LIN {X 0,Y 235.015,Z 372.088,A -85,B 0,C 180,E1 -19772.385,E2 -19772.385} C_VEL
LIN {X 0,Y 234.992,Z 371.84,A -85,B 0,C 180,E1 -19775.247,E2 -19775.247} C_VEL
LIN {X 0,Y 235.016,Z 371.83,A -85,B 0,C 180,E1 -19778.97,E2 -19778.97} C_VEL
LIN {X 0,Y 235.101,Z 371.824,A -85,B 0,C 180,E1 -19783.059,E2 -19783.059} C_VEL
LIN {X 0,Y 235.152,Z 371.812,A -85,B 0,C 180,E1 -19787.924,E2 -19787.924} C_VEL
LIN {X 0,Y 235.395,Z 371.781,A -85,B 0,C 180,E1 -19791.414,E2 -19791.414} C_VEL
LIN {X 0,Y 235.411,Z 371.788,A -85,B 0,C 180,E1 -19793.141,E2 -19793.141} C_VEL
LIN {X 0,Y 235.6,Z 371.755,A -85,B 0,C 180,E1 -19798.29,E2 -19798.29} C_VEL
LIN {X 0,Y 235.6,Z 371.755,A -85,B 0,C 180,E1 -19801.709,E2 -19801.709} C_VEL
LIN {X 0,Y 235.372,Z 371.79,A -85,B 0,C 180,E1 -19806.859,E2 -19806.859} C_VEL
LIN {X 0,Y 235.218,Z 371.808,A -85,B 0,C 180,E1 -19810.327,E2 -19810.327} C_VEL
LIN {X 0,Y 235.118,Z 371.831,A -85,B 0,C 180,E1 -19815.606,E2 -19815.606} C_VEL
LIN {X 0,Y 235.022,Z 371.874,A -85,B 0,C 180,E1 -19819.658,E2 -19819.658} C_VEL
LIN {X 0,Y 235.358,Z 373.616,A -85,B 0,C 180,E1 -19822.842,E2 -19822.842} C_VEL
LIN {X 0,Y 235.843,Z 375.925,A -85,B 0,C 180,E1 -19826.62,E2 -19826.62} C_VEL
LIN {X 0,Y 236.341,Z 378.635,A -85,B 0,C 180,E1 -19830.416,E2 -19830.416} C_VEL
LIN {X 0,Y 236.912,Z 381.747,A -85,B 0,C 180,E1 -19834.307,E2 -19834.307} C_VEL
LIN {X 0,Y 237.605,Z 385.363,A -85,B 0,C 180,E1 -19838.4,E2 -19838.4} C_VEL
LIN {X 0,Y 238.386,Z 389.338,A -85,B 0,C 180,E1 -19842.519,E2 -19842.519} C_VEL
LIN {X 0,Y 238.664,Z 390.728,A -85,B 0,C 180,E1 -19843.886,E2 -19843.886} C_VEL
LIN {X 0,Y 238.895,Z 392.241,A -85,B 0,C 180,E1 -19844.731,E2 -19844.731} C_VEL
LIN {X 0,Y 239.346,Z 395.314,A -85,B 0,C 180,E1 -19845.625,E2 -19845.625} C_VEL
LIN {X 0,Y 240.189,Z 400.855,A -85,B 0,C 180,E1 -19846.595,E2 -19846.595} C_VEL
LIN {X 0,Y 243.299,Z 415.71,A -85,B 0,C 180,E1 -19848.361,E2 -19848.361} C_VEL
LIN {X 0,Y 244.82,Z 420.413,A -85,B 0,C 180,E1 -19849.055,E2 -19849.055} C_VEL
LIN {X 0,Y 247.249,Z 433.501,A -85,B 0,C 180,E1 -19850.799,E2 -19850.799} C_VEL
LIN {X 0,Y 248.739,Z 446.866,A -85,B 0,C 180,E1 -19852.698,E2 -19852.698} C_VEL
LIN {X 0,Y 249.245,Z 459.354,A -85,B 0,C 180,E1 -19854.629,E2 -19854.629} C_VEL
LIN {X 0,Y 248.915,Z 463.831,A -85,B 0,C 180,E1 -19855.336,E2 -19855.336} C_VEL
LIN {X 0,Y 245.212,Z 476.724,A -85,B 0,C 180,E1 -19857.249,E2 -19857.249} C_VEL
LIN {X 0,Y 241.61,Z 488.325,A -85,B 0,C 180,E1 -19859.399,E2 -19859.399} C_VEL
LIN {X 0,Y 238.108,Z 498.941,A -85,B 0,C 180,E1 -19861.819,E2 -19861.819} C_VEL
LIN {X 0,Y 235.174,Z 507.913,A -85,B 0,C 180,E1 -19864.321,E2 -19864.321} C_VEL
LIN {X 0,Y 232.556,Z 515.567,A -85,B 0,C 180,E1 -19866.866,E2 -19866.866} C_VEL
LIN {X 0,Y 230.383,Z 522.077,A -85,B 0,C 180,E1 -19869.462,E2 -19869.462} C_VEL
LIN {X 0,Y 228.333,Z 528.833,A -85,B 0,C 180,E1 -19872.78,E2 -19872.78} C_VEL
LIN {X 0,Y 226.762,Z 534.808,A -85,B 0,C 180,E1 -19876.559,E2 -19876.559} C_VEL
LIN {X 0,Y 226.093,Z 538.041,A -85,B 0,C 180,E1 -19879.251,E2 -19879.251} C_VEL
LIN {X 0,Y 225.715,Z 541.228,A -85,B 0,C 180,E1 -19882.845,E2 -19882.845} C_VEL
LIN {X 0,Y 225.73,Z 543.137,A -85,B 0,C 180,E1 -19886.43,E2 -19886.43} C_VEL
LIN {X 0,Y 225.822,Z 543.621,A -85,B 0,C 180,E1 -19888.216,E2 -19888.216} C_VEL
LIN {X 0,Y 225.878,Z 543.785,A -85,B 0,C 180,E1 -19890,E2 -19890} C_VEL
LIN {X 0,Y 225.823,Z 543.616,A -85,B 0,C 180,E1 -19891.783,E2 -19891.783} C_VEL
LIN {X 0,Y 225.741,Z 542.321,A -85,B 0,C 180,E1 -19895.359,E2 -19895.359} C_VEL
LIN {X 0,Y 225.869,Z 539.762,A -85,B 0,C 180,E1 -19898.95,E2 -19898.95} C_VEL
LIN {X 0,Y 226.451,Z 535.904,A -85,B 0,C 180,E1 -19902.547,E2 -19902.547} C_VEL
LIN {X 0,Y 227.762,Z 530.665,A -85,B 0,C 180,E1 -19906.124,E2 -19906.124} C_VEL
LIN {X 0,Y 229.759,Z 523.911,A -85,B 0,C 180,E1 -19909.662,E2 -19909.662} C_VEL
LIN {X 0,Y 232.12,Z 516.601,A -85,B 0,C 180,E1 -19912.708,E2 -19912.708} C_VEL
LIN {X 0,Y 235.14,Z 507.788,A -85,B 0,C 180,E1 -19915.683,E2 -19915.683} C_VEL
LIN {X 0,Y 238.097,Z 498.791,A -85,B 0,C 180,E1 -19918.182,E2 -19918.182} C_VEL
LIN {X 0,Y 241.563,Z 488.144,A -85,B 0,C 180,E1 -19920.607,E2 -19920.607} C_VEL
LIN {X 0,Y 245.156,Z 476.511,A -85,B 0,C 180,E1 -19922.759,E2 -19922.759} C_VEL
LIN {X 0,Y 248.879,Z 463.799,A -85,B 0,C 180,E1 -19924.63,E2 -19924.63} C_VEL
LIN {X 0,Y 249.127,Z 457.221,A -85,B 0,C 180,E1 -19925.672,E2 -19925.672} C_VEL
LIN {X 0,Y 248.45,Z 444.428,A -85,B 0,C 180,E1 -19927.623,E2 -19927.623} C_VEL
LIN {X 0,Y 246.857,Z 431.262,A -85,B 0,C 180,E1 -19929.47,E2 -19929.47} C_VEL
LIN {X 0,Y 244.147,Z 418.018,A -85,B 0,C 180,E1 -19931.234,E2 -19931.234} C_VEL
LIN {X 0,Y 241.259,Z 411.166,A -85,B 0,C 180,E1 -19932.337,E2 -19932.337} C_VEL
LIN {X 0,Y 236.412,Z 401.706,A -85,B 0,C 180,E1 -19933.98,E2 -19933.98} C_VEL
LIN {X 0,Y 234.193,Z 397.541,A -85,B 0,C 180,E1 -19934.687,E2 -19934.687} C_VEL
LIN {X 0,Y 232.289,Z 394.258,A -85,B 0,C 180,E1 -19935.292,E2 -19935.292} C_VEL
LIN {X 0,Y 231.858,Z 392.833,A -85,B 0,C 180,E1 -19935.518,E2 -19935.518} C_VEL
LIN {X 0,Y 231.002,Z 388.18,A -85,B 0,C 180,E1 -19940.29,E2 -19940.29} C_VEL
LIN {X 0,Y 230.054,Z 383.593,A -85,B 0,C 180,E1 -19945.572,E2 -19945.572} C_VEL
LIN {X 0,Y 229.331,Z 379.702,A -85,B 0,C 180,E1 -19950.638,E2 -19950.638} C_VEL
LIN {X 0,Y 228.852,Z 377.106,A -85,B 0,C 180,E1 -19954.537,E2 -19954.537} C_VEL
LIN {X 0,Y 228.397,Z 374.912,A -85,B 0,C 180,E1 -19958.331,E2 -19958.331} C_VEL
LIN {X 0,Y 228.04,Z 372.704,A -85,B 0,C 180,E1 -19962.823,E2 -19962.823} C_VEL
LIN {X 0,Y 228.076,Z 372.692,A -85,B 0,C 180,E1 -19967.544,E2 -19967.544} C_VEL
LIN {X 0,Y 228.266,Z 372.671,A -85,B 0,C 180,E1 -19971.145,E2 -19971.145} C_VEL
LIN {X 0,Y 228.322,Z 372.663,A -85,B 0,C 180,E1 -19972.928,E2 -19972.928} C_VEL
LIN {X 0,Y 228.557,Z 372.636,A -85,B 0,C 180,E1 -19978.238,E2 -19978.238} C_VEL
LIN {X 0,Y 228.557,Z 372.635,A -85,B 0,C 180,E1 -19981.762,E2 -19981.762} C_VEL
LIN {X 0,Y 228.362,Z 372.658,A -85,B 0,C 180,E1 -19987.072,E2 -19987.072} C_VEL
LIN {X 0,Y 228.175,Z 372.681,A -85,B 0,C 180,E1 -19990.65,E2 -19990.65} C_VEL
LIN {X 0,Y 228.069,Z 372.694,A -85,B 0,C 180,E1 -19994.272,E2 -19994.272} C_VEL
LIN {X 0,Y 228.006,Z 372.701,A -85,B 0,C 180,E1 -19997.953,E2 -19997.953} C_VEL
LIN {X 0,Y 227.933,Z 372.716,A -85,B 0,C 180,E1 -20002.33,E2 -20002.33} C_VEL
LIN {X 0,Y 227.946,Z 372.773,A -85,B 0,C 180,E1 -20005.084,E2 -20005.084} C_VEL
LIN {X 0,Y 228.303,Z 374.704,A -85,B 0,C 180,E1 -20009.508,E2 -20009.508} C_VEL
LIN {X 0,Y 228.687,Z 376.954,A -85,B 0,C 180,E1 -20013.925,E2 -20013.925} C_VEL
LIN {X 0,Y 229.075,Z 379.212,A -85,B 0,C 180,E1 -20017.851,E2 -20017.851} C_VEL
LIN {X 0,Y 229.499,Z 382.119,A -85,B 0,C 180,E1 -20022.355,E2 -20022.355} C_VEL
LIN {X 0,Y 229.854,Z 384.793,A -85,B 0,C 180,E1 -20026.131,E2 -20026.131} C_VEL
LIN {X 0,Y 229.888,Z 385.286,A -85,B 0,C 180,E1 -20026.793,E2 -20026.793} C_VEL
LIN {X 0,Y 231.265,Z 388.595,A -85,B 0,C 180,E1 -20027.302,E2 -20027.302} C_VEL
LIN {X 0,Y 232.899,Z 390.912,A -85,B 0,C 180,E1 -20027.804,E2 -20027.804} C_VEL
LIN {X 0,Y 237.12,Z 399.072,A -85,B 0,C 180,E1 -20029.257,E2 -20029.257} C_VEL
LIN {X 0,Y 241.328,Z 409.168,A -85,B 0,C 180,E1 -20030.956,E2 -20030.956} C_VEL
LIN {X 0,Y 245.03,Z 420.57,A -85,B 0,C 180,E1 -20032.812,E2 -20032.812} C_VEL
LIN {X 0,Y 247.842,Z 432.547,A -85,B 0,C 180,E1 -20034.79,E2 -20034.79} C_VEL
LIN {X 0,Y 249.545,Z 443.432,A -85,B 0,C 180,E1 -20036.689,E2 -20036.689} C_VEL
LIN {X 0,Y 250.061,Z 449.138,A -85,B 0,C 180,E1 -20037.724,E2 -20037.724} C_VEL
LIN {X 0,Y 247.163,Z 460.518,A -85,B 0,C 180,E1 -20039.451,E2 -20039.451} C_VEL
LIN {X 0,Y 244.196,Z 470.062,A -85,B 0,C 180,E1 -20041.179,E2 -20041.179} C_VEL
LIN {X 0,Y 240.769,Z 480.693,A -85,B 0,C 180,E1 -20043.567,E2 -20043.567} C_VEL
LIN {X 0,Y 237.529,Z 489.516,A -85,B 0,C 180,E1 -20045.994,E2 -20045.994} C_VEL
LIN {X 0,Y 234.851,Z 496.873,A -85,B 0,C 180,E1 -20048.487,E2 -20048.487} C_VEL
LIN {X 0,Y 232.143,Z 503.98,A -85,B 0,C 180,E1 -20051.465,E2 -20051.465} C_VEL
LIN {X 0,Y 229.682,Z 510.385,A -85,B 0,C 180,E1 -20054.925,E2 -20054.925} C_VEL
LIN {X 0,Y 227.926,Z 515.224,A -85,B 0,C 180,E1 -20058.438,E2 -20058.438} C_VEL
LIN {X 0,Y 227.059,Z 517.955,A -85,B 0,C 180,E1 -20061.097,E2 -20061.097} C_VEL
LIN {X 0,Y 226.328,Z 520.408,A -85,B 0,C 180,E1 -20064.655,E2 -20064.655} C_VEL
LIN {X 0,Y 225.966,Z 521.628,A -85,B 0,C 180,E1 -20068.218,E2 -20068.218} C_VEL
LIN {X 0,Y 225.965,Z 521.649,A -85,B 0,C 180,E1 -20071.783,E2 -20071.783} C_VEL
LIN {X 0,Y 226.317,Z 520.472,A -85,B 0,C 180,E1 -20075.346,E2 -20075.346} C_VEL
LIN {X 0,Y 226.992,Z 518.066,A -85,B 0,C 180,E1 -20078.906,E2 -20078.906} C_VEL
LIN {X 0,Y 228.275,Z 514.344,A -85,B 0,C 180,E1 -20082.446,E2 -20082.446} C_VEL
LIN {X 0,Y 230.161,Z 509.188,A -85,B 0,C 180,E1 -20085.951,E2 -20085.951} C_VEL
LIN {X 0,Y 232.106,Z 504.242,A -85,B 0,C 180,E1 -20088.538,E2 -20088.538} C_VEL
LIN {X 0,Y 234.807,Z 497.263,A -85,B 0,C 180,E1 -20091.488,E2 -20091.488} C_VEL
LIN {X 0,Y 237.423,Z 489.902,A -85,B 0,C 180,E1 -20094.018,E2 -20094.018} C_VEL
LIN {X 0,Y 240.657,Z 481.158,A -85,B 0,C 180,E1 -20096.446,E2 -20096.446} C_VEL
LIN {X 0,Y 244.11,Z 470.614,A -85,B 0,C 180,E1 -20098.832,E2 -20098.832} C_VEL
LIN {X 0,Y 247.705,Z 458.972,A -85,B 0,C 180,E1 -20100.921,E2 -20100.921} C_VEL
LIN {X 0,Y 250.104,Z 449.936,A -85,B 0,C 180,E1 -20102.27,E2 -20102.27} C_VEL
LIN {X 0,Y 249.142,Z 440.073,A -85,B 0,C 180,E1 -20104.042,E2 -20104.042} C_VEL
LIN {X 0,Y 247.061,Z 428.423,A -85,B 0,C 180,E1 -20106.02,E2 -20106.02} C_VEL
LIN {X 0,Y 243.944,Z 416.811,A -85,B 0,C 180,E1 -20107.937,E2 -20107.937} C_VEL
LIN {X 0,Y 239.95,Z 405.345,A -85,B 0,C 180,E1 -20109.811,E2 -20109.811} C_VEL
LIN {X 0,Y 235.604,Z 396.058,A -85,B 0,C 180,E1 -20111.422,E2 -20111.422} C_VEL
LIN {X 0,Y 232.307,Z 389.929,A -85,B 0,C 180,E1 -20112.542,E2 -20112.542} C_VEL
LIN {X 0,Y 230.416,Z 386.973,A -85,B 0,C 180,E1 -20113.145,E2 -20113.145} C_VEL
LIN {X 0,Y 229.888,Z 385.248,A -85,B 0,C 180,E1 -20113.423,E2 -20113.423} C_VEL
LIN {X 0,Y 229.514,Z 382.232,A -85,B 0,C 180,E1 -20117.649,E2 -20117.649} C_VEL
LIN {X 0,Y 229.081,Z 379.34,A -85,B 0,C 180,E1 -20122.151,E2 -20122.151} C_VEL
LIN {X 0,Y 228.711,Z 376.86,A -85,B 0,C 180,E1 -20126.418,E2 -20126.418} C_VEL
LIN {X 0,Y 228.339,Z 374.816,A -85,B 0,C 180,E1 -20130.497,E2 -20130.497} C_VEL
LIN {X 0,Y 227.964,Z 372.715,A -85,B 0,C 180,E1 -20135.344,E2 -20135.344} C_VEL
LIN {X 0,Y 227.966,Z 372.711,A -85,B 0,C 180,E1 -20138.287,E2 -20138.287} C_VEL
LIN {X 0,Y 228.039,Z 372.701,A -85,B 0,C 180,E1 -20142.825,E2 -20142.825} C_VEL
LIN {X 0,Y 228.099,Z 372.692,A -85,B 0,C 180,E1 -20147.544,E2 -20147.544} C_VEL
LIN {X 0,Y 228.33,Z 372.661,A -85,B 0,C 180,E1 -20151.147,E2 -20151.147} C_VEL
LIN {X 0,Y 228.363,Z 372.665,A -85,B 0,C 180,E1 -20152.928,E2 -20152.928} C_VEL
LIN {X 0,Y 228.559,Z 372.632,A -85,B 0,C 180,E1 -20158.238,E2 -20158.238} C_VEL
LIN {X 0,Y 228.558,Z 372.632,A -85,B 0,C 180,E1 -20161.762,E2 -20161.762} C_VEL
LIN {X 0,Y 228.322,Z 372.666,A -85,B 0,C 180,E1 -20167.072,E2 -20167.072} C_VEL
LIN {X 0,Y 228.154,Z 372.687,A -85,B 0,C 180,E1 -20170.65,E2 -20170.65} C_VEL
LIN {X 0,Y 228.069,Z 372.699,A -85,B 0,C 180,E1 -20174.271,E2 -20174.271} C_VEL
LIN {X 0,Y 228.05,Z 372.792,A -85,B 0,C 180,E1 -20177.184,E2 -20177.184} C_VEL
LIN {X 0,Y 228.434,Z 374.987,A -85,B 0,C 180,E1 -20181.665,E2 -20181.665} C_VEL
LIN {X 0,Y 228.886,Z 377.188,A -85,B 0,C 180,E1 -20185.459,E2 -20185.459} C_VEL
LIN {X 0,Y 229.361,Z 379.796,A -85,B 0,C 180,E1 -20189.358,E2 -20189.358} C_VEL
LIN {X 0,Y 230.068,Z 383.667,A -85,B 0,C 180,E1 -20194.433,E2 -20194.433} C_VEL
LIN {X 0,Y 230.591,Z 386.357,A -85,B 0,C 180,E1 -20197.585,E2 -20197.585} C_VEL
LIN {X 0,Y 231.386,Z 390.359,A -85,B 0,C 180,E1 -20201.929,E2 -20201.929} C_VEL
LIN {X 0,Y 231.861,Z 392.923,A -85,B 0,C 180,E1 -20204.48,E2 -20204.48} C_VEL
LIN {X 0,Y 233.212,Z 396.174,A -85,B 0,C 180,E1 -20204.951,E2 -20204.951} C_VEL
LIN {X 0,Y 234.925,Z 398.782,A -85,B 0,C 180,E1 -20205.478,E2 -20205.478} C_VEL
LIN {X 0,Y 241.608,Z 411.82,A -85,B 0,C 180,E1 -20207.727,E2 -20207.727} C_VEL
LIN {X 0,Y 243.299,Z 415.71,A -85,B 0,C 180,E1 -20208.361,E2 -20208.361} C_VEL
LIN {X 0,Y 244.001,Z 419.161,A -85,B 0,C 180,E1 -20208.777,E2 -20208.777} C_VEL
LIN {X 0,Y 244.156,Z 424.646,A -85,B 0,C 180,E1 -20209.308,E2 -20209.308} C_VEL
LIN {X 0,Y 242.658,Z 437.693,A -85,B 0,C 180,E1 -20210.463,E2 -20210.463} C_VEL
LIN {X 0,Y 242.29,Z 443.055,A -85,B 0,C 180,E1 -20211.089,E2 -20211.089} C_VEL
LIN {X 0,Y 242.378,Z 444.76,A -85,B 0,C 180,E1 -20211.333,E2 -20211.333} C_VEL
LIN {X 0,Y 242.974,Z 457.515,A -85,B 0,C 180,E1 -20213.361,E2 -20213.361} C_VEL
LIN {X 0,Y 242.891,Z 463.353,A -85,B 0,C 180,E1 -20214.347,E2 -20214.347} C_VEL
LIN {X 0,Y 240.378,Z 472.767,A -85,B 0,C 180,E1 -20215.749,E2 -20215.749} C_VEL
LIN {X 0,Y 236.768,Z 483.974,A -85,B 0,C 180,E1 -20217.703,E2 -20217.703} C_VEL
LIN {X 0,Y 232.983,Z 495.257,A -85,B 0,C 180,E1 -20220.15,E2 -20220.15} C_VEL
LIN {X 0,Y 229.694,Z 504.738,A -85,B 0,C 180,E1 -20222.68,E2 -20222.68} C_VEL
LIN {X 0,Y 226.471,Z 514.036,A -85,B 0,C 180,E1 -20225.72,E2 -20225.72} C_VEL
LIN {X 0,Y 223.63,Z 521.714,A -85,B 0,C 180,E1 -20228.813,E2 -20228.813} C_VEL
LIN {X 0,Y 221.33,Z 528.944,A -85,B 0,C 180,E1 -20232.486,E2 -20232.486} C_VEL
LIN {X 0,Y 219.779,Z 534.456,A -85,B 0,C 180,E1 -20236.123,E2 -20236.123} C_VEL
LIN {X 0,Y 219.069,Z 537.692,A -85,B 0,C 180,E1 -20238.902,E2 -20238.902} C_VEL
LIN {X 0,Y 218.628,Z 540.881,A -85,B 0,C 180,E1 -20242.612,E2 -20242.612} C_VEL
LIN {X 0,Y 218.64,Z 542.791,A -85,B 0,C 180,E1 -20246.314,E2 -20246.314} C_VEL
LIN {X 0,Y 218.809,Z 543.44,A -85,B 0,C 180,E1 -20250,E2 -20250} C_VEL
LIN {X 0,Y 218.731,Z 543.271,A -85,B 0,C 180,E1 -20251.841,E2 -20251.841} C_VEL
LIN {X 0,Y 218.647,Z 541.974,A -85,B 0,C 180,E1 -20255.533,E2 -20255.533} C_VEL
LIN {X 0,Y 218.796,Z 539.413,A -85,B 0,C 180,E1 -20259.242,E2 -20259.242} C_VEL
LIN {X 0,Y 219.467,Z 535.553,A -85,B 0,C 180,E1 -20262.953,E2 -20262.953} C_VEL
LIN {X 0,Y 220.854,Z 530.309,A -85,B 0,C 180,E1 -20266.642,E2 -20266.642} C_VEL
LIN {X 0,Y 222.991,Z 523.55,A -85,B 0,C 180,E1 -20270.285,E2 -20270.285} C_VEL
LIN {X 0,Y 225.527,Z 516.235,A -85,B 0,C 180,E1 -20273.411,E2 -20273.411} C_VEL
LIN {X 0,Y 228.695,Z 507.412,A -85,B 0,C 180,E1 -20276.462,E2 -20276.462} C_VEL
LIN {X 0,Y 232.34,Z 496.75,A -85,B 0,C 180,E1 -20279.442,E2 -20279.442} C_VEL
LIN {X 0,Y 236.114,Z 485.771,A -85,B 0,C 180,E1 -20281.893,E2 -20281.893} C_VEL
LIN {X 0,Y 239.579,Z 474.902,A -85,B 0,C 180,E1 -20283.874,E2 -20283.874} C_VEL
LIN {X 0,Y 242.646,Z 464.741,A -85,B 0,C 180,E1 -20285.4,E2 -20285.4} C_VEL
LIN {X 0,Y 242.904,Z 455.67,A -85,B 0,C 180,E1 -20286.896,E2 -20286.896} C_VEL
LIN {X 0,Y 242.101,Z 442.227,A -85,B 0,C 180,E1 -20288.997,E2 -20288.997} C_VEL
LIN {X 0,Y 240.271,Z 428.605,A -85,B 0,C 180,E1 -20290.97,E2 -20290.97} C_VEL
LIN {X 0,Y 238.358,Z 420.17,A -85,B 0,C 180,E1 -20292.189,E2 -20292.189} C_VEL
LIN {X 0,Y 233.484,Z 409.417,A -85,B 0,C 180,E1 -20294.135,E2 -20294.135} C_VEL
LIN {X 0,Y 229.654,Z 402.034,A -85,B 0,C 180,E1 -20295.519,E2 -20295.519} C_VEL
LIN {X 0,Y 227.202,Z 397.587,A -85,B 0,C 180,E1 -20296.359,E2 -20296.359} C_VEL
LIN {X 0,Y 225.212,Z 394.558,A -85,B 0,C 180,E1 -20297.027,E2 -20297.027} C_VEL
LIN {X 0,Y 224.567,Z 392.591,A -85,B 0,C 180,E1 -20297.333,E2 -20297.333} C_VEL
LIN {X 0,Y 223.899,Z 389.135,A -85,B 0,C 180,E1 -20301.114,E2 -20301.114} C_VEL
LIN {X 0,Y 223.225,Z 385.48,A -85,B 0,C 180,E1 -20305.479,E2 -20305.479} C_VEL
LIN {X 0,Y 222.612,Z 382.328,A -85,B 0,C 180,E1 -20309.66,E2 -20309.66} C_VEL
LIN {X 0,Y 222.129,Z 379.615,A -85,B 0,C 180,E1 -20313.708,E2 -20313.708} C_VEL
LIN {X 0,Y 221.694,Z 377.313,A -85,B 0,C 180,E1 -20317.641,E2 -20317.641} C_VEL
LIN {X 0,Y 221.213,Z 374.557,A -85,B 0,C 180,E1 -20323.386,E2 -20323.386} C_VEL
LIN {X 0,Y 221.007,Z 373.575,A -85,B 0,C 180,E1 -20326.202,E2 -20326.202} C_VEL
LIN {X 0,Y 221.204,Z 373.549,A -85,B 0,C 180,E1 -20330.86,E2 -20330.86} C_VEL
LIN {X 0,Y 221.141,Z 373.558,A -85,B 0,C 180,E1 -20334.529,E2 -20334.529} C_VEL
LIN {X 0,Y 221.515,Z 373.513,A -85,B 0,C 180,E1 -20338.182,E2 -20338.182} C_VEL
LIN {X 0,Y 221.515,Z 373.513,A -85,B 0,C 180,E1 -20341.818,E2 -20341.818} C_VEL
LIN {X 0,Y 221.299,Z 373.536,A -85,B 0,C 180,E1 -20347.298,E2 -20347.298} C_VEL
LIN {X 0,Y 221.12,Z 373.558,A -85,B 0,C 180,E1 -20350.994,E2 -20350.994} C_VEL
LIN {X 0,Y 221.02,Z 373.58,A -85,B 0,C 180,E1 -20356.63,E2 -20356.63} C_VEL
LIN {X 0,Y 220.907,Z 373.635,A -85,B 0,C 180,E1 -20362.198,E2 -20362.198} C_VEL
LIN {X 0,Y 221.21,Z 375.203,A -85,B 0,C 180,E1 -20366.41,E2 -20366.41} C_VEL
LIN {X 0,Y 221.553,Z 377.285,A -85,B 0,C 180,E1 -20371.076,E2 -20371.076} C_VEL
LIN {X 0,Y 221.881,Z 379.157,A -85,B 0,C 180,E1 -20374.761,E2 -20374.761} C_VEL
LIN {X 0,Y 222.167,Z 380.841,A -85,B 0,C 180,E1 -20377.735,E2 -20377.735} C_VEL
LIN {X 0,Y 222.487,Z 383.225,A -85,B 0,C 180,E1 -20381.557,E2 -20381.557} C_VEL
LIN {X 0,Y 222.921,Z 385.725,A -85,B 0,C 180,E1 -20385.023,E2 -20385.023} C_VEL
LIN {X 0,Y 224.353,Z 388.977,A -85,B 0,C 180,E1 -20385.576,E2 -20385.576} C_VEL
LIN {X 0,Y 225.895,Z 390.967,A -85,B 0,C 180,E1 -20386.081,E2 -20386.081} C_VEL
LIN {X 0,Y 228.091,Z 394.897,A -85,B 0,C 180,E1 -20386.876,E2 -20386.876} C_VEL
LIN {X 0,Y 232.253,Z 403.056,A -85,B 0,C 180,E1 -20388.464,E2 -20388.464} C_VEL
LIN {X 0,Y 236.139,Z 412.811,A -85,B 0,C 180,E1 -20390.195,E2 -20390.195} C_VEL
LIN {X 0,Y 239.781,Z 425.003,A -85,B 0,C 180,E1 -20392.314,E2 -20392.314} C_VEL
LIN {X 0,Y 242.16,Z 436.585,A -85,B 0,C 180,E1 -20394.353,E2 -20394.353} C_VEL
LIN {X 0,Y 243.584,Z 447.83,A -85,B 0,C 180,E1 -20396.434,E2 -20396.434} C_VEL
LIN {X 0,Y 243.841,Z 450.945,A -85,B 0,C 180,E1 -20397.029,E2 -20397.029} C_VEL
LIN {X 0,Y 240.444,Z 463.235,A -85,B 0,C 180,E1 -20398.991,E2 -20398.991} C_VEL
LIN {X 0,Y 237.391,Z 472.402,A -85,B 0,C 180,E1 -20400.759,E2 -20400.759} C_VEL
LIN {X 0,Y 233.843,Z 482.688,A -85,B 0,C 180,E1 -20403.204,E2 -20403.204} C_VEL
LIN {X 0,Y 230.544,Z 491.22,A -85,B 0,C 180,E1 -20405.698,E2 -20405.698} C_VEL
LIN {X 0,Y 227.842,Z 498.346,A -85,B 0,C 180,E1 -20408.275,E2 -20408.275} C_VEL
LIN {X 0,Y 225.428,Z 504.335,A -85,B 0,C 180,E1 -20410.892,E2 -20410.892} C_VEL
LIN {X 0,Y 222.828,Z 510.737,A -85,B 0,C 180,E1 -20414.449,E2 -20414.449} C_VEL
LIN {X 0,Y 220.983,Z 515.572,A -85,B 0,C 180,E1 -20418.07,E2 -20418.07} C_VEL
LIN {X 0,Y 220.039,Z 518.302,A -85,B 0,C 180,E1 -20420.811,E2 -20420.811} C_VEL
LIN {X 0,Y 219.277,Z 520.753,A -85,B 0,C 180,E1 -20424.482,E2 -20424.482} C_VEL
LIN {X 0,Y 218.901,Z 521.973,A -85,B 0,C 180,E1 -20428.16,E2 -20428.16} C_VEL
LIN {X 0,Y 218.901,Z 521.992,A -85,B 0,C 180,E1 -20431.84,E2 -20431.84} C_VEL
LIN {X 0,Y 219.264,Z 520.817,A -85,B 0,C 180,E1 -20435.518,E2 -20435.518} C_VEL
LIN {X 0,Y 219.994,Z 518.411,A -85,B 0,C 180,E1 -20439.192,E2 -20439.192} C_VEL
LIN {X 0,Y 221.334,Z 514.691,A -85,B 0,C 180,E1 -20442.843,E2 -20442.843} C_VEL
LIN {X 0,Y 223.318,Z 509.539,A -85,B 0,C 180,E1 -20446.454,E2 -20446.454} C_VEL
LIN {X 0,Y 225.394,Z 504.593,A -85,B 0,C 180,E1 -20449.111,E2 -20449.111} C_VEL
LIN {X 0,Y 227.826,Z 498.662,A -85,B 0,C 180,E1 -20451.727,E2 -20451.727} C_VEL
LIN {X 0,Y 230.467,Z 491.601,A -85,B 0,C 180,E1 -20454.311,E2 -20454.311} C_VEL
LIN {X 0,Y 233.754,Z 483.145,A -85,B 0,C 180,E1 -20456.807,E2 -20456.807} C_VEL
LIN {X 0,Y 237.292,Z 472.951,A -85,B 0,C 180,E1 -20459.255,E2 -20459.255} C_VEL
LIN {X 0,Y 241.004,Z 461.602,A -85,B 0,C 180,E1 -20461.417,E2 -20461.417} C_VEL
LIN {X 0,Y 243.852,Z 451.485,A -85,B 0,C 180,E1 -20463.008,E2 -20463.008} C_VEL
LIN {X 0,Y 242.964,Z 441.531,A -85,B 0,C 180,E1 -20464.878,E2 -20464.878} C_VEL
LIN {X 0,Y 241.093,Z 430.386,A -85,B 0,C 180,E1 -20466.875,E2 -20466.875} C_VEL
LIN {X 0,Y 238.141,Z 418.907,A -85,B 0,C 180,E1 -20468.886,E2 -20468.886} C_VEL
LIN {X 0,Y 234.361,Z 408.023,A -85,B 0,C 180,E1 -20470.791,E2 -20470.791} C_VEL
LIN {X 0,Y 230.227,Z 398.868,A -85,B 0,C 180,E1 -20472.5,E2 -20472.5} C_VEL
LIN {X 0,Y 227.695,Z 394.359,A -85,B 0,C 180,E1 -20473.421,E2 -20473.421} C_VEL
LIN {X 0,Y 225.391,Z 390.245,A -85,B 0,C 180,E1 -20474.252,E2 -20474.252} C_VEL
LIN {X 0,Y 223.394,Z 387.223,A -85,B 0,C 180,E1 -20474.939,E2 -20474.939} C_VEL
LIN {X 0,Y 222.858,Z 385.533,A -85,B 0,C 180,E1 -20475.2,E2 -20475.2} C_VEL
LIN {X 0,Y 222.415,Z 382.777,A -85,B 0,C 180,E1 -20479.321,E2 -20479.321} C_VEL
LIN {X 0,Y 222.114,Z 380.498,A -85,B 0,C 180,E1 -20483.045,E2 -20483.045} C_VEL
LIN {X 0,Y 221.697,Z 378.158,A -85,B 0,C 180,E1 -20487.39,E2 -20487.39} C_VEL
LIN {X 0,Y 221.37,Z 376.21,A -85,B 0,C 180,E1 -20491.561,E2 -20491.561} C_VEL
LIN {X 0,Y 221.076,Z 374.534,A -85,B 0,C 180,E1 -20495.589,E2 -20495.589} C_VEL
LIN {X 0,Y 220.907,Z 373.589,A -85,B 0,C 180,E1 -20498.539,E2 -20498.539} C_VEL
LIN {X 0,Y 221.021,Z 373.58,A -85,B 0,C 180,E1 -20503.37,E2 -20503.37} C_VEL
LIN {X 0,Y 221.121,Z 373.561,A -85,B 0,C 180,E1 -20509.006,E2 -20509.006} C_VEL
LIN {X 0,Y 221.3,Z 373.542,A -85,B 0,C 180,E1 -20512.702,E2 -20512.702} C_VEL
LIN {X 0,Y 221.517,Z 373.509,A -85,B 0,C 180,E1 -20518.182,E2 -20518.182} C_VEL
LIN {X 0,Y 221.516,Z 373.509,A -85,B 0,C 180,E1 -20521.818,E2 -20521.818} C_VEL
LIN {X 0,Y 221.258,Z 373.545,A -85,B 0,C 180,E1 -20527.299,E2 -20527.299} C_VEL
LIN {X 0,Y 221.091,Z 373.566,A -85,B 0,C 180,E1 -20530.995,E2 -20530.995} C_VEL
LIN {X 0,Y 221.053,Z 373.71,A -85,B 0,C 180,E1 -20534.264,E2 -20534.264} C_VEL
LIN {X 0,Y 221.33,Z 375.494,A -85,B 0,C 180,E1 -20538.514,E2 -20538.514} C_VEL
LIN {X 0,Y 221.79,Z 377.884,A -85,B 0,C 180,E1 -20543.227,E2 -20543.227} C_VEL
LIN {X 0,Y 222.306,Z 380.616,A -85,B 0,C 180,E1 -20547.723,E2 -20547.723} C_VEL
LIN {X 0,Y 222.877,Z 383.955,A -85,B 0,C 180,E1 -20552.416,E2 -20552.416} C_VEL
LIN {X 0,Y 223.327,Z 386.006,A -85,B 0,C 180,E1 -20555.093,E2 -20555.093} C_VEL
LIN {X 0,Y 224.163,Z 390.192,A -85,B 0,C 180,E1 -20559.995,E2 -20559.995} C_VEL
LIN {X 0,Y 224.612,Z 392.731,A -85,B 0,C 180,E1 -20562.656,E2 -20562.656} C_VEL
LIN {X 0,Y 225.846,Z 395.783,A -85,B 0,C 180,E1 -20563.128,E2 -20563.128} C_VEL
LIN {X 0,Y 227.793,Z 398.516,A -85,B 0,C 180,E1 -20563.767,E2 -20563.767} C_VEL
LIN {X 0,Y 229.995,Z 402.508,A -85,B 0,C 180,E1 -20564.525,E2 -20564.525} C_VEL
LIN {X 0,Y 235.969,Z 414.575,A -85,B 0,C 180,E1 -20566.762,E2 -20566.762} C_VEL
LIN {X 0,Y 239.107,Z 422.363,A -85,B 0,C 180,E1 -20568.109,E2 -20568.109} C_VEL
LIN {X 0,Y 241.46,Z 435.947,A -85,B 0,C 180,E1 -20570.036,E2 -20570.036} C_VEL
LIN {X 0,Y 242.378,Z 444.76,A -85,B 0,C 180,E1 -20571.333,E2 -20571.333} C_VEL
LIN {X 0,Y 242.2,Z 449.904,A -85,B 0,C 180,E1 -20572.033,E2 -20572.033} C_VEL
LIN {X 0,Y 240.982,Z 455.164,A -85,B 0,C 180,E1 -20572.642,E2 -20572.642} C_VEL
LIN {X 0,Y 237.023,Z 465.548,A -85,B 0,C 180,E1 -20573.808,E2 -20573.808} C_VEL
LIN {X 0,Y 234.538,Z 472.177,A -85,B 0,C 180,E1 -20574.737,E2 -20574.737} C_VEL
LIN {X 0,Y 230.749,Z 483.565,A -85,B 0,C 180,E1 -20576.754,E2 -20576.754} C_VEL
LIN {X 0,Y 226.779,Z 494.869,A -85,B 0,C 180,E1 -20579.246,E2 -20579.246} C_VEL
LIN {X 0,Y 223.052,Z 505.147,A -85,B 0,C 180,E1 -20582.068,E2 -20582.068} C_VEL
LIN {X 0,Y 219.957,Z 513.669,A -85,B 0,C 180,E1 -20584.953,E2 -20584.953} C_VEL
LIN {X 0,Y 216.944,Z 521.354,A -85,B 0,C 180,E1 -20588.127,E2 -20588.127} C_VEL
LIN {X 0,Y 214.584,Z 528.339,A -85,B 0,C 180,E1 -20591.768,E2 -20591.768} C_VEL
LIN {X 0,Y 212.811,Z 534.103,A -85,B 0,C 180,E1 -20595.659,E2 -20595.659} C_VEL
LIN {X 0,Y 212.034,Z 537.343,A -85,B 0,C 180,E1 -20598.529,E2 -20598.529} C_VEL
LIN {X 0,Y 211.564,Z 540.534,A -85,B 0,C 180,E1 -20602.364,E2 -20602.364} C_VEL
LIN {X 0,Y 211.555,Z 542.446,A -85,B 0,C 180,E1 -20606.19,E2 -20606.19} C_VEL
LIN {X 0,Y 211.741,Z 543.096,A -85,B 0,C 180,E1 -20610,E2 -20610} C_VEL
LIN {X 0,Y 211.556,Z 542.432,A -85,B 0,C 180,E1 -20613.809,E2 -20613.809} C_VEL
LIN {X 0,Y 211.604,Z 540.505,A -85,B 0,C 180,E1 -20617.634,E2 -20617.634} C_VEL
LIN {X 0,Y 212.034,Z 537.299,A -85,B 0,C 180,E1 -20621.471,E2 -20621.471} C_VEL
LIN {X 0,Y 213.131,Z 532.758,A -85,B 0,C 180,E1 -20625.296,E2 -20625.296} C_VEL
LIN {X 0,Y 215,Z 526.771,A -85,B 0,C 180,E1 -20629.08,E2 -20629.08} C_VEL
LIN {X 0,Y 217.704,Z 519.186,A -85,B 0,C 180,E1 -20632.792,E2 -20632.792} C_VEL
LIN {X 0,Y 220.853,Z 511.035,A -85,B 0,C 180,E1 -20635.948,E2 -20635.948} C_VEL
LIN {X 0,Y 224.295,Z 501.5,A -85,B 0,C 180,E1 -20638.954,E2 -20638.954} C_VEL
LIN {X 0,Y 228.013,Z 491.102,A -85,B 0,C 180,E1 -20641.6,E2 -20641.6} C_VEL
LIN {X 0,Y 231.766,Z 480.135,A -85,B 0,C 180,E1 -20643.862,E2 -20643.862} C_VEL
LIN {X 0,Y 235.668,Z 468.293,A -85,B 0,C 180,E1 -20645.816,E2 -20645.816} C_VEL
LIN {X 0,Y 236.618,Z 464.25,A -85,B 0,C 180,E1 -20646.444,E2 -20646.444} C_VEL
LIN {X 0,Y 236.633,Z 451.835,A -85,B 0,C 180,E1 -20648.587,E2 -20648.587} C_VEL
LIN {X 0,Y 235.727,Z 439.76,A -85,B 0,C 180,E1 -20650.514,E2 -20650.514} C_VEL
LIN {X 0,Y 233.98,Z 427.62,A -85,B 0,C 180,E1 -20652.343,E2 -20652.343} C_VEL
LIN {X 0,Y 233.406,Z 424.687,A -85,B 0,C 180,E1 -20652.789,E2 -20652.789} C_VEL
LIN {X 0,Y 228.952,Z 414.241,A -85,B 0,C 180,E1 -20654.777,E2 -20654.777} C_VEL
LIN {X 0,Y 224.884,Z 406.132,A -85,B 0,C 180,E1 -20656.411,E2 -20656.411} C_VEL
LIN {X 0,Y 222.805,Z 402.27,A -85,B 0,C 180,E1 -20657.222,E2 -20657.222} C_VEL
LIN {X 0,Y 220.578,Z 398.166,A -85,B 0,C 180,E1 -20658.061,E2 -20658.061} C_VEL
LIN {X 0,Y 218.004,Z 394.342,A -85,B 0,C 180,E1 -20658.999,E2 -20658.999} C_VEL
LIN {X 0,Y 217.343,Z 392.346,A -85,B 0,C 180,E1 -20659.326,E2 -20659.326} C_VEL
LIN {X 0,Y 216.503,Z 388.25,A -85,B 0,C 180,E1 -20664.246,E2 -20664.246} C_VEL
LIN {X 0,Y 215.92,Z 384.942,A -85,B 0,C 180,E1 -20668.615,E2 -20668.615} C_VEL
LIN {X 0,Y 215.407,Z 382.13,A -85,B 0,C 180,E1 -20672.821,E2 -20672.821} C_VEL
LIN {X 0,Y 214.967,Z 379.733,A -85,B 0,C 180,E1 -20676.901,E2 -20676.901} C_VEL
LIN {X 0,Y 214.441,Z 376.861,A -85,B 0,C 180,E1 -20682.845,E2 -20682.845} C_VEL
LIN {X 0,Y 214.146,Z 375.405,A -85,B 0,C 180,E1 -20686.719,E2 -20686.719} C_VEL
LIN {X 0,Y 214.125,Z 374.43,A -85,B 0,C 180,E1 -20689.952,E2 -20689.952} C_VEL
LIN {X 0,Y 214.197,Z 374.425,A -85,B 0,C 180,E1 -20692.459,E2 -20692.459} C_VEL
LIN {X 0,Y 214.448,Z 374.392,A -85,B 0,C 180,E1 -20698.122,E2 -20698.122} C_VEL
LIN {X 0,Y 214.553,Z 374.376,A -85,B 0,C 180,E1 -20700,E2 -20700} C_VEL
LIN {X 0,Y 214.449,Z 374.393,A -85,B 0,C 180,E1 -20701.878,E2 -20701.878} C_VEL
LIN {X 0,Y 214.239,Z 374.414,A -85,B 0,C 180,E1 -20707.54,E2 -20707.54} C_VEL
LIN {X 0,Y 214.051,Z 374.437,A -85,B 0,C 180,E1 -20711.362,E2 -20711.362} C_VEL
LIN {X 0,Y 213.937,Z 374.453,A -85,B 0,C 180,E1 -20715.237,E2 -20715.237} C_VEL
LIN {X 0,Y 213.907,Z 374.57,A -85,B 0,C 180,E1 -20718.744,E2 -20718.744} C_VEL
LIN {X 0,Y 214.127,Z 375.932,A -85,B 0,C 180,E1 -20723.218,E2 -20723.218} C_VEL
LIN {X 0,Y 214.449,Z 377.648,A -85,B 0,C 180,E1 -20727.766,E2 -20727.766} C_VEL
LIN {X 0,Y 214.738,Z 379.404,A -85,B 0,C 180,E1 -20731.686,E2 -20731.686} C_VEL
LIN {X 0,Y 215.114,Z 381.61,A -85,B 0,C 180,E1 -20736.021,E2 -20736.021} C_VEL
LIN {X 0,Y 215.52,Z 384.338,A -85,B 0,C 180,E1 -20740.707,E2 -20740.707} C_VEL
LIN {X 0,Y 215.73,Z 385.826,A -85,B 0,C 180,E1 -20742.976,E2 -20742.976} C_VEL
LIN {X 0,Y 217.078,Z 388.94,A -85,B 0,C 180,E1 -20743.549,E2 -20743.549} C_VEL
LIN {X 0,Y 219.117,Z 391.477,A -85,B 0,C 180,E1 -20744.277,E2 -20744.277} C_VEL
LIN {X 0,Y 221.152,Z 395.096,A -85,B 0,C 180,E1 -20745.079,E2 -20745.079} C_VEL
LIN {X 0,Y 224.867,Z 401.925,A -85,B 0,C 180,E1 -20746.573,E2 -20746.573} C_VEL
LIN {X 0,Y 228.125,Z 409.01,A -85,B 0,C 180,E1 -20748.011,E2 -20748.011} C_VEL
LIN {X 0,Y 231.525,Z 418.426,A -85,B 0,C 180,E1 -20749.792,E2 -20749.792} C_VEL
LIN {X 0,Y 234.634,Z 430.334,A -85,B 0,C 180,E1 -20751.987,E2 -20751.987} C_VEL
LIN {X 0,Y 236.569,Z 441.3,A -85,B 0,C 180,E1 -20754.052,E2 -20754.052} C_VEL
LIN {X 0,Y 237.601,Z 452.294,A -85,B 0,C 180,E1 -20756.219,E2 -20756.219} C_VEL
LIN {X 0,Y 234.412,Z 463.652,A -85,B 0,C 180,E1 -20758.101,E2 -20758.101} C_VEL
LIN {X 0,Y 231.242,Z 472.806,A -85,B 0,C 180,E1 -20759.902,E2 -20759.902} C_VEL
LIN {X 0,Y 227.545,Z 483.073,A -85,B 0,C 180,E1 -20762.4,E2 -20762.4} C_VEL
LIN {X 0,Y 224.109,Z 491.59,A -85,B 0,C 180,E1 -20764.953,E2 -20764.953} C_VEL
LIN {X 0,Y 221.233,Z 498.708,A -85,B 0,C 180,E1 -20767.591,E2 -20767.591} C_VEL
LIN {X 0,Y 218.739,Z 504.689,A -85,B 0,C 180,E1 -20770.284,E2 -20770.284} C_VEL
LIN {X 0,Y 216.574,Z 509.669,A -85,B 0,C 180,E1 -20773.019,E2 -20773.019} C_VEL
LIN {X 0,Y 214.451,Z 514.885,A -85,B 0,C 180,E1 -20776.738,E2 -20776.738} C_VEL
LIN {X 0,Y 213.02,Z 518.649,A -85,B 0,C 180,E1 -20780.505,E2 -20780.505} C_VEL
LIN {X 0,Y 212.208,Z 521.099,A -85,B 0,C 180,E1 -20784.298,E2 -20784.298} C_VEL
LIN {X 0,Y 211.838,Z 522.317,A -85,B 0,C 180,E1 -20788.099,E2 -20788.099} C_VEL
LIN {X 0,Y 211.838,Z 522.336,A -85,B 0,C 180,E1 -20791.901,E2 -20791.901} C_VEL
LIN {X 0,Y 212.196,Z 521.162,A -85,B 0,C 180,E1 -20795.703,E2 -20795.703} C_VEL
LIN {X 0,Y 212.988,Z 518.756,A -85,B 0,C 180,E1 -20799.497,E2 -20799.497} C_VEL
LIN {X 0,Y 214.413,Z 515.037,A -85,B 0,C 180,E1 -20803.265,E2 -20803.265} C_VEL
LIN {X 0,Y 216.497,Z 509.89,A -85,B 0,C 180,E1 -20806.988,E2 -20806.988} C_VEL
LIN {X 0,Y 218.709,Z 504.944,A -85,B 0,C 180,E1 -20809.719,E2 -20809.719} C_VEL
LIN {X 0,Y 221.204,Z 499.022,A -85,B 0,C 180,E1 -20812.412,E2 -20812.412} C_VEL
LIN {X 0,Y 224.005,Z 491.969,A -85,B 0,C 180,E1 -20815.06,E2 -20815.06} C_VEL
LIN {X 0,Y 227.437,Z 483.523,A -85,B 0,C 180,E1 -20817.614,E2 -20817.614} C_VEL
LIN {X 0,Y 231.128,Z 473.349,A -85,B 0,C 180,E1 -20820.114,E2 -20820.114} C_VEL
LIN {X 0,Y 234.656,Z 463.172,A -85,B 0,C 180,E1 -20822.115,E2 -20822.115} C_VEL
LIN {X 0,Y 237.685,Z 452.678,A -85,B 0,C 180,E1 -20823.831,E2 -20823.831} C_VEL
LIN {X 0,Y 236.692,Z 441.785,A -85,B 0,C 180,E1 -20825.991,E2 -20825.991} C_VEL
LIN {X 0,Y 234.654,Z 429.981,A -85,B 0,C 180,E1 -20828.209,E2 -20828.209} C_VEL
LIN {X 0,Y 231.611,Z 418.598,A -85,B 0,C 180,E1 -20830.323,E2 -20830.323} C_VEL
LIN {X 0,Y 228.39,Z 409.509,A -85,B 0,C 180,E1 -20832.034,E2 -20832.034} C_VEL
LIN {X 0,Y 223.911,Z 399.909,A -85,B 0,C 180,E1 -20834.01,E2 -20834.01} C_VEL
LIN {X 0,Y 220.782,Z 394.594,A -85,B 0,C 180,E1 -20835.227,E2 -20835.227} C_VEL
LIN {X 0,Y 218.588,Z 390.746,A -85,B 0,C 180,E1 -20836.086,E2 -20836.086} C_VEL
LIN {X 0,Y 216.407,Z 387.79,A -85,B 0,C 180,E1 -20836.89,E2 -20836.89} C_VEL
LIN {X 0,Y 215.688,Z 385.745,A -85,B 0,C 180,E1 -20837.268,E2 -20837.268} C_VEL
LIN {X 0,Y 215.334,Z 383.029,A -85,B 0,C 180,E1 -20841.675,E2 -20841.675} C_VEL
LIN {X 0,Y 214.911,Z 380.551,A -85,B 0,C 180,E1 -20846.225,E2 -20846.225} C_VEL
LIN {X 0,Y 214.579,Z 378.505,A -85,B 0,C 180,E1 -20850.574,E2 -20850.574} C_VEL
LIN {X 0,Y 214.297,Z 376.774,A -85,B 0,C 180,E1 -20854.764,E2 -20854.764} C_VEL
LIN {X 0,Y 214.055,Z 375.38,A -85,B 0,C 180,E1 -20858.828,E2 -20858.828} C_VEL
LIN {X 0,Y 213.948,Z 374.456,A -85,B 0,C 180,E1 -20862.804,E2 -20862.804} C_VEL
LIN {X 0,Y 213.985,Z 374.456,A -85,B 0,C 180,E1 -20866.708,E2 -20866.708} C_VEL
LIN {X 0,Y 214.201,Z 374.424,A -85,B 0,C 180,E1 -20870.557,E2 -20870.557} C_VEL
LIN {X 0,Y 214.115,Z 374.431,A -85,B 0,C 180,E1 -20874.349,E2 -20874.349} C_VEL
LIN {X 0,Y 214.451,Z 374.389,A -85,B 0,C 180,E1 -20878.122,E2 -20878.122} C_VEL
LIN {X 0,Y 214.555,Z 374.385,A -85,B 0,C 180,E1 -20880,E2 -20880} C_VEL
LIN {X 0,Y 214.449,Z 374.39,A -85,B 0,C 180,E1 -20881.878,E2 -20881.878} C_VEL
LIN {X 0,Y 214.198,Z 374.423,A -85,B 0,C 180,E1 -20887.541,E2 -20887.541} C_VEL
LIN {X 0,Y 214.129,Z 374.456,A -85,B 0,C 180,E1 -20890.052,E2 -20890.052} C_VEL
LIN {X 0,Y 214.317,Z 376.177,A -85,B 0,C 180,E1 -20895.209,E2 -20895.209} C_VEL
LIN {X 0,Y 214.577,Z 377.836,A -85,B 0,C 180,E1 -20899.118,E2 -20899.118} C_VEL
LIN {X 0,Y 215.052,Z 380.219,A -85,B 0,C 180,E1 -20903.785,E2 -20903.785} C_VEL
LIN {X 0,Y 215.551,Z 382.935,A -85,B 0,C 180,E1 -20908.317,E2 -20908.317} C_VEL
LIN {X 0,Y 216.002,Z 385.656,A -85,B 0,C 180,E1 -20912.225,E2 -20912.225} C_VEL
LIN {X 0,Y 216.528,Z 388.33,A -85,B 0,C 180,E1 -20915.762,E2 -20915.762} C_VEL
LIN {X 0,Y 217.336,Z 392.431,A -85,B 0,C 180,E1 -20920.628,E2 -20920.628} C_VEL
LIN {X 0,Y 218.672,Z 395.624,A -85,B 0,C 180,E1 -20921.182,E2 -20921.182} C_VEL
LIN {X 0,Y 220.699,Z 398.467,A -85,B 0,C 180,E1 -20921.911,E2 -20921.911} C_VEL
LIN {X 0,Y 222.931,Z 402.445,A -85,B 0,C 180,E1 -20922.748,E2 -20922.748} C_VEL
LIN {X 0,Y 228.181,Z 412.47,A -85,B 0,C 180,E1 -20924.825,E2 -20924.825} C_VEL
LIN {X 0,Y 232.78,Z 422.968,A -85,B 0,C 180,E1 -20926.84,E2 -20926.84} C_VEL
LIN {X 0,Y 234.071,Z 427.479,A -85,B 0,C 180,E1 -20927.601,E2 -20927.601} C_VEL
LIN {X 0,Y 235.819,Z 439.857,A -85,B 0,C 180,E1 -20929.459,E2 -20929.459} C_VEL
LIN {X 0,Y 236.713,Z 452.198,A -85,B 0,C 180,E1 -20931.428,E2 -20931.428} C_VEL
LIN {X 0,Y 236.669,Z 464.532,A -85,B 0,C 180,E1 -20933.565,E2 -20933.565} C_VEL
LIN {X 0,Y 234.538,Z 472.177,A -85,B 0,C 180,E1 -20934.737,E2 -20934.737} C_VEL
LIN {X 0,Y 232.472,Z 476.923,A -85,B 0,C 180,E1 -20935.439,E2 -20935.439} C_VEL
LIN {X 0,Y 227.446,Z 484.423,A -85,B 0,C 180,E1 -20936.468,E2 -20936.468} C_VEL
LIN {X 0,Y 222.342,Z 491.522,A -85,B 0,C 180,E1 -20937.653,E2 -20937.653} C_VEL
LIN {X 0,Y 220.193,Z 495.636,A -85,B 0,C 180,E1 -20938.595,E2 -20938.595} C_VEL
LIN {X 0,Y 216.476,Z 505.417,A -85,B 0,C 180,E1 -20941.388,E2 -20941.388} C_VEL
LIN {X 0,Y 212.986,Z 514.484,A -85,B 0,C 180,E1 -20944.597,E2 -20944.597} C_VEL
LIN {X 0,Y 210.307,Z 520.995,A -85,B 0,C 180,E1 -20947.399,E2 -20947.399} C_VEL
LIN {X 0,Y 207.598,Z 528.454,A -85,B 0,C 180,E1 -20951.424,E2 -20951.424} C_VEL
LIN {X 0,Y 205.862,Z 533.751,A -85,B 0,C 180,E1 -20955.164,E2 -20955.164} C_VEL
LIN {X 0,Y 204.995,Z 536.992,A -85,B 0,C 180,E1 -20958.129,E2 -20958.129} C_VEL
LIN {X 0,Y 204.477,Z 540.186,A -85,B 0,C 180,E1 -20962.098,E2 -20962.098} C_VEL
LIN {X 0,Y 204.472,Z 542.101,A -85,B 0,C 180,E1 -20966.058,E2 -20966.058} C_VEL
LIN {X 0,Y 204.674,Z 542.752,A -85,B 0,C 180,E1 -20970,E2 -20970} C_VEL
LIN {X 0,Y 204.472,Z 542.087,A -85,B 0,C 180,E1 -20973.942,E2 -20973.942} C_VEL
LIN {X 0,Y 204.525,Z 540.157,A -85,B 0,C 180,E1 -20977.9,E2 -20977.9} C_VEL
LIN {X 0,Y 204.994,Z 536.948,A -85,B 0,C 180,E1 -20981.871,E2 -20981.871} C_VEL
LIN {X 0,Y 206.202,Z 532.404,A -85,B 0,C 180,E1 -20985.823,E2 -20985.823} C_VEL
LIN {X 0,Y 208.235,Z 526.414,A -85,B 0,C 180,E1 -20989.725,E2 -20989.725} C_VEL
LIN {X 0,Y 211.069,Z 518.822,A -85,B 0,C 180,E1 -20993.551,E2 -20993.551} C_VEL
LIN {X 0,Y 214.395,Z 510.663,A -85,B 0,C 180,E1 -20996.791,E2 -20996.791} C_VEL
LIN {X 0,Y 218.125,Z 500.815,A -85,B 0,C 180,E1 -20999.961,E2 -20999.961} C_VEL
LIN {X 0,Y 221.941,Z 490.704,A -85,B 0,C 180,E1 -21002.57,E2 -21002.57} C_VEL
LIN {X 0,Y 225.825,Z 479.712,A -85,B 0,C 180,E1 -21004.88,E2 -21004.88} C_VEL
LIN {X 0,Y 229.781,Z 468.204,A -85,B 0,C 180,E1 -21006.805,E2 -21006.805} C_VEL
LIN {X 0,Y 230.439,Z 465.25,A -85,B 0,C 180,E1 -21007.3,E2 -21007.3} C_VEL
LIN {X 0,Y 230.589,Z 453.39,A -85,B 0,C 180,E1 -21009.436,E2 -21009.436} C_VEL
LIN {X 0,Y 229.857,Z 441.13,A -85,B 0,C 180,E1 -21011.489,E2 -21011.489} C_VEL
LIN {X 0,Y 228.32,Z 429.524,A -85,B 0,C 180,E1 -21013.347,E2 -21013.347} C_VEL
LIN {X 0,Y 226.818,Z 424.834,A -85,B 0,C 180,E1 -21014.231,E2 -21014.231} C_VEL
LIN {X 0,Y 221.74,Z 413.219,A -85,B 0,C 180,E1 -21016.636,E2 -21016.636} C_VEL
LIN {X 0,Y 218.426,Z 406.904,A -85,B 0,C 180,E1 -21018.059,E2 -21018.059} C_VEL
LIN {X 0,Y 215.613,Z 401.89,A -85,B 0,C 180,E1 -21019.238,E2 -21019.238} C_VEL
LIN {X 0,Y 213.552,Z 398.084,A -85,B 0,C 180,E1 -21020.09,E2 -21020.09} C_VEL
LIN {X 0,Y 210.841,Z 394.319,A -85,B 0,C 180,E1 -21021.165,E2 -21021.165} C_VEL
LIN {X 0,Y 210.02,Z 392.111,A -85,B 0,C 180,E1 -21021.599,E2 -21021.599} C_VEL
LIN {X 0,Y 209.222,Z 387.88,A -85,B 0,C 180,E1 -21027.117,E2 -21027.117} C_VEL
LIN {X 0,Y 208.691,Z 384.664,A -85,B 0,C 180,E1 -21031.87,E2 -21031.87} C_VEL
LIN {X 0,Y 208.209,Z 382.182,A -85,B 0,C 180,E1 -21036.106,E2 -21036.106} C_VEL
LIN {X 0,Y 207.719,Z 379.612,A -85,B 0,C 180,E1 -21041.327,E2 -21041.327} C_VEL
LIN {X 0,Y 207.538,Z 378.37,A -85,B 0,C 180,E1 -21044.282,E2 -21044.282} C_VEL
LIN {X 0,Y 207.336,Z 376.419,A -85,B 0,C 180,E1 -21050.243,E2 -21050.243} C_VEL
LIN {X 0,Y 207.091,Z 375.559,A -85,B 0,C 180,E1 -21054.157,E2 -21054.157} C_VEL
LIN {X 0,Y 207.385,Z 375.271,A -85,B 0,C 180,E1 -21058.058,E2 -21058.058} C_VEL
LIN {X 0,Y 207.518,Z 375.252,A -85,B 0,C 180,E1 -21060,E2 -21060} C_VEL
LIN {X 0,Y 207.385,Z 375.273,A -85,B 0,C 180,E1 -21061.942,E2 -21061.942} C_VEL
LIN {X 0,Y 207.182,Z 375.292,A -85,B 0,C 180,E1 -21067.799,E2 -21067.799} C_VEL
LIN {X 0,Y 206.986,Z 375.317,A -85,B 0,C 180,E1 -21071.755,E2 -21071.755} C_VEL
LIN {X 0,Y 206.981,Z 375.875,A -85,B 0,C 180,E1 -21075.762,E2 -21075.762} C_VEL
LIN {X 0,Y 207.112,Z 376.869,A -85,B 0,C 180,E1 -21079.837,E2 -21079.837} C_VEL
LIN {X 0,Y 207.333,Z 378.149,A -85,B 0,C 180,E1 -21084.002,E2 -21084.002} C_VEL
LIN {X 0,Y 207.62,Z 379.764,A -85,B 0,C 180,E1 -21088.344,E2 -21088.344} C_VEL
LIN {X 0,Y 207.932,Z 381.727,A -85,B 0,C 180,E1 -21092.738,E2 -21092.738} C_VEL
LIN {X 0,Y 208.252,Z 383.304,A -85,B 0,C 180,E1 -21095.91,E2 -21095.91} C_VEL
LIN {X 0,Y 208.651,Z 386.12,A -85,B 0,C 180,E1 -21100.739,E2 -21100.739} C_VEL
LIN {X 0,Y 209.988,Z 389.18,A -85,B 0,C 180,E1 -21101.367,E2 -21101.367} C_VEL
LIN {X 0,Y 212.183,Z 391.92,A -85,B 0,C 180,E1 -21102.235,E2 -21102.235} C_VEL
LIN {X 0,Y 214.396,Z 395.653,A -85,B 0,C 180,E1 -21103.181,E2 -21103.181} C_VEL
LIN {X 0,Y 215.477,Z 397.384,A -85,B 0,C 180,E1 -21103.634,E2 -21103.634} C_VEL
LIN {X 0,Y 218.525,Z 402.959,A -85,B 0,C 180,E1 -21104.97,E2 -21104.97} C_VEL
LIN {X 0,Y 222.275,Z 410.722,A -85,B 0,C 180,E1 -21106.727,E2 -21106.727} C_VEL
LIN {X 0,Y 225.755,Z 420.322,A -85,B 0,C 180,E1 -21108.681,E2 -21108.681} C_VEL
LIN {X 0,Y 228.703,Z 431.994,A -85,B 0,C 180,E1 -21110.969,E2 -21110.969} C_VEL
LIN {X 0,Y 230.509,Z 443.029,A -85,B 0,C 180,E1 -21113.163,E2 -21113.163} C_VEL
LIN {X 0,Y 231.379,Z 453.222,A -85,B 0,C 180,E1 -21115.276,E2 -21115.276} C_VEL
LIN {X 0,Y 231.01,Z 455.744,A -85,B 0,C 180,E1 -21115.736,E2 -21115.736} C_VEL
LIN {X 0,Y 227.326,Z 467.259,A -85,B 0,C 180,E1 -21117.771,E2 -21117.771} C_VEL
LIN {X 0,Y 223.808,Z 476.816,A -85,B 0,C 180,E1 -21119.839,E2 -21119.839} C_VEL
LIN {X 0,Y 220.004,Z 486.438,A -85,B 0,C 180,E1 -21122.406,E2 -21122.406} C_VEL
LIN {X 0,Y 216.624,Z 494.463,A -85,B 0,C 180,E1 -21125.054,E2 -21125.054} C_VEL
LIN {X 0,Y 213.834,Z 501.197,A -85,B 0,C 180,E1 -21127.792,E2 -21127.792} C_VEL
LIN {X 0,Y 210.464,Z 508.449,A -85,B 0,C 180,E1 -21131.504,E2 -21131.504} C_VEL
LIN {X 0,Y 208.018,Z 514.038,A -85,B 0,C 180,E1 -21135.322,E2 -21135.322} C_VEL
LIN {X 0,Y 206.688,Z 517.286,A -85,B 0,C 180,E1 -21138.228,E2 -21138.228} C_VEL
LIN {X 0,Y 205.535,Z 520.377,A -85,B 0,C 180,E1 -21142.139,E2 -21142.139} C_VEL
LIN {X 0,Y 204.914,Z 522.204,A -85,B 0,C 180,E1 -21146.067,E2 -21146.067} C_VEL
LIN {X 0,Y 204.698,Z 522.821,A -85,B 0,C 180,E1 -21150,E2 -21150} C_VEL
LIN {X 0,Y 204.91,Z 522.244,A -85,B 0,C 180,E1 -21153.934,E2 -21153.934} C_VEL
LIN {X 0,Y 205.487,Z 520.462,A -85,B 0,C 180,E1 -21157.863,E2 -21157.863} C_VEL
LIN {X 0,Y 206.665,Z 517.411,A -85,B 0,C 180,E1 -21161.774,E2 -21161.774} C_VEL
LIN {X 0,Y 208.53,Z 512.999,A -85,B 0,C 180,E1 -21165.642,E2 -21165.642} C_VEL
LIN {X 0,Y 211.185,Z 507.065,A -85,B 0,C 180,E1 -21169.438,E2 -21169.438} C_VEL
LIN {X 0,Y 214.235,Z 500.471,A -85,B 0,C 180,E1 -21172.673,E2 -21172.673} C_VEL
LIN {X 0,Y 217.045,Z 493.594,A -85,B 0,C 180,E1 -21175.407,E2 -21175.407} C_VEL
LIN {X 0,Y 220.552,Z 485.377,A -85,B 0,C 180,E1 -21178.036,E2 -21178.036} C_VEL
LIN {X 0,Y 224.367,Z 475.54,A -85,B 0,C 180,E1 -21180.598,E2 -21180.598} C_VEL
LIN {X 0,Y 228.347,Z 464.648,A -85,B 0,C 180,E1 -21182.852,E2 -21182.852} C_VEL
LIN {X 0,Y 231.227,Z 455.273,A -85,B 0,C 180,E1 -21184.468,E2 -21184.468} C_VEL
LIN {X 0,Y 231.463,Z 452.847,A -85,B 0,C 180,E1 -21184.933,E2 -21184.933} C_VEL
LIN {X 0,Y 230.468,Z 441.958,A -85,B 0,C 180,E1 -21187.186,E2 -21187.186} C_VEL
LIN {X 0,Y 228.627,Z 431.299,A -85,B 0,C 180,E1 -21189.304,E2 -21189.304} C_VEL
LIN {X 0,Y 225.582,Z 419.604,A -85,B 0,C 180,E1 -21191.606,E2 -21191.606} C_VEL
LIN {X 0,Y 221.536,Z 408.862,A -85,B 0,C 180,E1 -21193.823,E2 -21193.823} C_VEL
LIN {X 0,Y 217.009,Z 400.032,A -85,B 0,C 180,E1 -21195.895,E2 -21195.895} C_VEL
LIN {X 0,Y 214.423,Z 395.668,A -85,B 0,C 180,E1 -21196.987,E2 -21196.987} C_VEL
LIN {X 0,Y 212.191,Z 391.947,A -85,B 0,C 180,E1 -21197.942,E2 -21197.942} C_VEL
LIN {X 0,Y 209.334,Z 388.041,A -85,B 0,C 180,E1 -21199.104,E2 -21199.104} C_VEL
LIN {X 0,Y 208.616,Z 386.024,A -85,B 0,C 180,E1 -21199.491,E2 -21199.491} C_VEL
LIN {X 0,Y 208.258,Z 383.423,A -85,B 0,C 180,E1 -21204.089,E2 -21204.089} C_VEL
LIN {X 0,Y 207.922,Z 381.649,A -85,B 0,C 180,E1 -21207.676,E2 -21207.676} C_VEL
LIN {X 0,Y 207.65,Z 379.893,A -85,B 0,C 180,E1 -21211.716,E2 -21211.716} C_VEL
LIN {X 0,Y 207.326,Z 378.194,A -85,B 0,C 180,E1 -21216.244,E2 -21216.244} C_VEL
LIN {X 0,Y 207.13,Z 376.992,A -85,B 0,C 180,E1 -21220.165,E2 -21220.165} C_VEL
LIN {X 0,Y 206.988,Z 376.003,A -85,B 0,C 180,E1 -21224.238,E2 -21224.238} C_VEL
LIN {X 0,Y 206.988,Z 375.319,A -85,B 0,C 180,E1 -21228.245,E2 -21228.245} C_VEL
LIN {X 0,Y 207.183,Z 375.296,A -85,B 0,C 180,E1 -21232.201,E2 -21232.201} C_VEL
LIN {X 0,Y 207.387,Z 375.268,A -85,B 0,C 180,E1 -21238.058,E2 -21238.058} C_VEL
LIN {X 0,Y 207.519,Z 375.262,A -85,B 0,C 180,E1 -21240,E2 -21240} C_VEL
LIN {X 0,Y 207.386,Z 375.269,A -85,B 0,C 180,E1 -21241.942,E2 -21241.942} C_VEL
LIN {X 0,Y 207.127,Z 375.635,A -85,B 0,C 180,E1 -21245.842,E2 -21245.842} C_VEL
LIN {X 0,Y 207.367,Z 376.494,A -85,B 0,C 180,E1 -21249.756,E2 -21249.756} C_VEL
LIN {X 0,Y 207.563,Z 378.48,A -85,B 0,C 180,E1 -21255.716,E2 -21255.716} C_VEL
LIN {X 0,Y 207.812,Z 380.201,A -85,B 0,C 180,E1 -21259.766,E2 -21259.766} C_VEL
LIN {X 0,Y 208.277,Z 382.534,A -85,B 0,C 180,E1 -21264.344,E2 -21264.344} C_VEL
LIN {X 0,Y 208.761,Z 385.253,A -85,B 0,C 180,E1 -21268.918,E2 -21268.918} C_VEL
LIN {X 0,Y 209.216,Z 387.961,A -85,B 0,C 180,E1 -21272.88,E2 -21272.88} C_VEL
LIN {X 0,Y 209.817,Z 391.116,A -85,B 0,C 180,E1 -21277.079,E2 -21277.079} C_VEL
LIN {X 0,Y 210.085,Z 392.327,A -85,B 0,C 180,E1 -21278.387,E2 -21278.387} C_VEL
LIN {X 0,Y 211.452,Z 395.448,A -85,B 0,C 180,E1 -21279.007,E2 -21279.007} C_VEL
LIN {X 0,Y 213.618,Z 398.223,A -85,B 0,C 180,E1 -21279.851,E2 -21279.851} C_VEL
LIN {X 0,Y 215.743,Z 402.106,A -85,B 0,C 180,E1 -21280.733,E2 -21280.733} C_VEL
LIN {X 0,Y 217.267,Z 404.868,A -85,B 0,C 180,E1 -21281.383,E2 -21281.383} C_VEL
LIN {X 0,Y 220.082,Z 410.018,A -85,B 0,C 180,E1 -21282.564,E2 -21282.564} C_VEL
LIN {X 0,Y 224.323,Z 418.933,A -85,B 0,C 180,E1 -21284.488,E2 -21284.488} C_VEL
LIN {X 0,Y 228.09,Z 428.272,A -85,B 0,C 180,E1 -21286.393,E2 -21286.393} C_VEL
LIN {X 0,Y 229.577,Z 437.432,A -85,B 0,C 180,E1 -21287.866,E2 -21287.866} C_VEL
LIN {X 0,Y 230.626,Z 451.639,A -85,B 0,C 180,E1 -21290.212,E2 -21290.212} C_VEL
LIN {X 0,Y 230.567,Z 464.037,A -85,B 0,C 180,E1 -21292.437,E2 -21292.437} C_VEL
LIN {X 0,Y 230.307,Z 466.779,A -85,B 0,C 180,E1 -21292.937,E2 -21292.937} C_VEL
LIN {X 0,Y 226.285,Z 478.852,A -85,B 0,C 180,E1 -21294.93,E2 -21294.93} C_VEL
LIN {X 0,Y 221.99,Z 490.887,A -85,B 0,C 180,E1 -21297.438,E2 -21297.438} C_VEL
LIN {X 0,Y 220.193,Z 495.636,A -85,B 0,C 180,E1 -21298.595,E2 -21298.595} C_VEL
LIN {X 0,Y 218.098,Z 499.692,A -85,B 0,C 180,E1 -21299.598,E2 -21299.598} C_VEL
LIN {X 0,Y 213.134,Z 505.899,A -85,B 0,C 180,E1 -21301.156,E2 -21301.156} C_VEL
LIN {X 0,Y 208.171,Z 511.707,A -85,B 0,C 180,E1 -21302.871,E2 -21302.871} C_VEL
LIN {X 0,Y 206.121,Z 514.99,A -85,B 0,C 180,E1 -21304.103,E2 -21304.103} C_VEL
LIN {X 0,Y 202.891,Z 522.569,A -85,B 0,C 180,E1 -21307.602,E2 -21307.602} C_VEL
LIN {X 0,Y 200.328,Z 529.316,A -85,B 0,C 180,E1 -21311.594,E2 -21311.594} C_VEL
LIN {X 0,Y 198.566,Z 534.55,A -85,B 0,C 180,E1 -21315.655,E2 -21315.655} C_VEL
LIN {X 0,Y 197.632,Z 538.405,A -85,B 0,C 180,E1 -21319.758,E2 -21319.758} C_VEL
LIN {X 0,Y 197.373,Z 540.956,A -85,B 0,C 180,E1 -21323.868,E2 -21323.868} C_VEL
LIN {X 0,Y 197.468,Z 542.24,A -85,B 0,C 180,E1 -21327.96,E2 -21327.96} C_VEL
LIN {X 0,Y 197.585,Z 542.407,A -85,B 0,C 180,E1 -21330,E2 -21330} C_VEL
LIN {X 0,Y 197.393,Z 541.741,A -85,B 0,C 180,E1 -21334.083,E2 -21334.083} C_VEL
LIN {X 0,Y 197.448,Z 539.808,A -85,B 0,C 180,E1 -21338.185,E2 -21338.185} C_VEL
LIN {X 0,Y 197.974,Z 536.596,A -85,B 0,C 180,E1 -21342.298,E2 -21342.298} C_VEL
LIN {X 0,Y 199.303,Z 532.051,A -85,B 0,C 180,E1 -21346.386,E2 -21346.386} C_VEL
LIN {X 0,Y 201.495,Z 526.058,A -85,B 0,C 180,E1 -21350.413,E2 -21350.413} C_VEL
LIN {X 0,Y 204.488,Z 518.459,A -85,B 0,C 180,E1 -21354.357,E2 -21354.357} C_VEL
LIN {X 0,Y 207.982,Z 510.292,A -85,B 0,C 180,E1 -21357.686,E2 -21357.686} C_VEL
LIN {X 0,Y 211.324,Z 501.941,A -85,B 0,C 180,E1 -21360.475,E2 -21360.475} C_VEL
LIN {X 0,Y 215.218,Z 492.106,A -85,B 0,C 180,E1 -21363.16,E2 -21363.16} C_VEL
LIN {X 0,Y 219.594,Z 480.367,A -85,B 0,C 180,E1 -21365.738,E2 -21365.738} C_VEL
LIN {X 0,Y 224.136,Z 467.591,A -85,B 0,C 180,E1 -21367.928,E2 -21367.928} C_VEL
LIN {X 0,Y 224.597,Z 456.939,A -85,B 0,C 180,E1 -21369.963,E2 -21369.963} C_VEL
LIN {X 0,Y 224.14,Z 443.749,A -85,B 0,C 180,E1 -21372.309,E2 -21372.309} C_VEL
LIN {X 0,Y 222.95,Z 433.074,A -85,B 0,C 180,E1 -21374.116,E2 -21374.116} C_VEL
LIN {X 0,Y 221.876,Z 429.272,A -85,B 0,C 180,E1 -21374.867,E2 -21374.867} C_VEL
LIN {X 0,Y 216.687,Z 416.746,A -85,B 0,C 180,E1 -21377.645,E2 -21377.645} C_VEL
LIN {X 0,Y 211.74,Z 407.144,A -85,B 0,C 180,E1 -21379.977,E2 -21379.977} C_VEL
LIN {X 0,Y 209,Z 402.369,A -85,B 0,C 180,E1 -21381.223,E2 -21381.223} C_VEL
LIN {X 0,Y 206.687,Z 398.522,A -85,B 0,C 180,E1 -21382.262,E2 -21382.262} C_VEL
LIN {X 0,Y 205.922,Z 397.322,A -85,B 0,C 180,E1 -21382.602,E2 -21382.602} C_VEL
LIN {X 0,Y 203.648,Z 394.249,A -85,B 0,C 180,E1 -21383.609,E2 -21383.609} C_VEL
LIN {X 0,Y 202.717,Z 391.848,A -85,B 0,C 180,E1 -21384.118,E2 -21384.118} C_VEL
LIN {X 0,Y 202.166,Z 388.715,A -85,B 0,C 180,E1 -21388.571,E2 -21388.571} C_VEL
LIN {X 0,Y 201.686,Z 385.881,A -85,B 0,C 180,E1 -21393.064,E2 -21393.064} C_VEL
LIN {X 0,Y 201.242,Z 383.507,A -85,B 0,C 180,E1 -21397.409,E2 -21397.409} C_VEL
LIN {X 0,Y 200.9,Z 381.527,A -85,B 0,C 180,E1 -21401.649,E2 -21401.649} C_VEL
LIN {X 0,Y 200.622,Z 379.929,A -85,B 0,C 180,E1 -21405.806,E2 -21405.806} C_VEL
LIN {X 0,Y 200.557,Z 378.642,A -85,B 0,C 180,E1 -21409.909,E2 -21409.909} C_VEL
LIN {X 0,Y 200.331,Z 377.725,A -85,B 0,C 180,E1 -21413.959,E2 -21413.959} C_VEL
LIN {X 0,Y 200.494,Z 377.002,A -85,B 0,C 180,E1 -21417.992,E2 -21417.992} C_VEL
LIN {X 0,Y 200.584,Z 376.774,A -85,B 0,C 180,E1 -21420,E2 -21420} C_VEL
LIN {X 0,Y 200.129,Z 376.753,A -85,B 0,C 180,E1 -21424.028,E2 -21424.028} C_VEL
LIN {X 0,Y 200.232,Z 376.847,A -85,B 0,C 180,E1 -21428.071,E2 -21428.071} C_VEL
LIN {X 0,Y 200.128,Z 377.302,A -85,B 0,C 180,E1 -21432.164,E2 -21432.164} C_VEL
LIN {X 0,Y 200.203,Z 378.026,A -85,B 0,C 180,E1 -21436.31,E2 -21436.31} C_VEL
LIN {X 0,Y 200.321,Z 379.046,A -85,B 0,C 180,E1 -21440.539,E2 -21440.539} C_VEL
LIN {X 0,Y 200.541,Z 380.388,A -85,B 0,C 180,E1 -21444.869,E2 -21444.869} C_VEL
LIN {X 0,Y 200.817,Z 382.07,A -85,B 0,C 180,E1 -21449.338,E2 -21449.338} C_VEL
LIN {X 0,Y 201.169,Z 384.145,A -85,B 0,C 180,E1 -21453.985,E2 -21453.985} C_VEL
LIN {X 0,Y 201.476,Z 386.286,A -85,B 0,C 180,E1 -21458.176,E2 -21458.176} C_VEL
LIN {X 0,Y 202.762,Z 389.229,A -85,B 0,C 180,E1 -21458.853,E2 -21458.853} C_VEL
LIN {X 0,Y 205.3,Z 392.265,A -85,B 0,C 180,E1 -21459.968,E2 -21459.968} C_VEL
LIN {X 0,Y 207.496,Z 396.027,A -85,B 0,C 180,E1 -21461.014,E2 -21461.014} C_VEL
LIN {X 0,Y 208.707,Z 397.818,A -85,B 0,C 180,E1 -21461.562,E2 -21461.562} C_VEL
LIN {X 0,Y 211.878,Z 403.343,A -85,B 0,C 180,E1 -21463.063,E2 -21463.063} C_VEL
LIN {X 0,Y 215.709,Z 410.816,A -85,B 0,C 180,E1 -21464.963,E2 -21464.963} C_VEL
LIN {X 0,Y 219.429,Z 420.326,A -85,B 0,C 180,E1 -21467.11,E2 -21467.11} C_VEL
LIN {X 0,Y 222.262,Z 431.073,A -85,B 0,C 180,E1 -21469.367,E2 -21469.367} C_VEL
LIN {X 0,Y 224.154,Z 441.846,A -85,B 0,C 180,E1 -21471.614,E2 -21471.614} C_VEL
LIN {X 0,Y 225.196,Z 452.702,A -85,B 0,C 180,E1 -21473.959,E2 -21473.959} C_VEL
LIN {X 0,Y 225.188,Z 456.194,A -85,B 0,C 180,E1 -21474.721,E2 -21474.721} C_VEL
LIN {X 0,Y 221.377,Z 467.675,A -85,B 0,C 180,E1 -21476.795,E2 -21476.795} C_VEL
LIN {X 0,Y 217.694,Z 477.21,A -85,B 0,C 180,E1 -21478.899,E2 -21478.899} C_VEL
LIN {X 0,Y 213.755,Z 486.814,A -85,B 0,C 180,E1 -21481.527,E2 -21481.527} C_VEL
LIN {X 0,Y 209.673,Z 496.002,A -85,B 0,C 180,E1 -21484.683,E2 -21484.683} C_VEL
LIN {X 0,Y 206.337,Z 503.528,A -85,B 0,C 180,E1 -21487.996,E2 -21487.996} C_VEL
LIN {X 0,Y 202.998,Z 510.376,A -85,B 0,C 180,E1 -21491.845,E2 -21491.845} C_VEL
LIN {X 0,Y 200.658,Z 515.582,A -85,B 0,C 180,E1 -21495.808,E2 -21495.808} C_VEL
LIN {X 0,Y 199.03,Z 519.342,A -85,B 0,C 180,E1 -21499.831,E2 -21499.831} C_VEL
LIN {X 0,Y 198.088,Z 521.791,A -85,B 0,C 180,E1 -21503.89,E2 -21503.89} C_VEL
LIN {X 0,Y 197.693,Z 523.006,A -85,B 0,C 180,E1 -21507.963,E2 -21507.963} C_VEL
LIN {X 0,Y 197.693,Z 523.025,A -85,B 0,C 180,E1 -21512.038,E2 -21512.038} C_VEL
LIN {X 0,Y 198.09,Z 521.851,A -85,B 0,C 180,E1 -21516.11,E2 -21516.11} C_VEL
LIN {X 0,Y 198.99,Z 519.446,A -85,B 0,C 180,E1 -21520.172,E2 -21520.172} C_VEL
LIN {X 0,Y 200.628,Z 515.728,A -85,B 0,C 180,E1 -21524.195,E2 -21524.195} C_VEL
LIN {X 0,Y 202.929,Z 510.59,A -85,B 0,C 180,E1 -21528.162,E2 -21528.162} C_VEL
LIN {X 0,Y 206.323,Z 503.805,A -85,B 0,C 180,E1 -21532.006,E2 -21532.006} C_VEL
LIN {X 0,Y 209.487,Z 496.584,A -85,B 0,C 180,E1 -21535.234,E2 -21535.234} C_VEL
LIN {X 0,Y 213.023,Z 488.682,A -85,B 0,C 180,E1 -21538.043,E2 -21538.043} C_VEL
LIN {X 0,Y 216.947,Z 479.448,A -85,B 0,C 180,E1 -21540.679,E2 -21540.679} C_VEL
LIN {X 0,Y 220.944,Z 469.286,A -85,B 0,C 180,E1 -21543.007,E2 -21543.007} C_VEL
LIN {X 0,Y 224.87,Z 457.634,A -85,B 0,C 180,E1 -21545.177,E2 -21545.177} C_VEL
LIN {X 0,Y 225.369,Z 455.479,A -85,B 0,C 180,E1 -21545.549,E2 -21545.549} C_VEL
LIN {X 0,Y 224.483,Z 443.69,A -85,B 0,C 180,E1 -21548.13,E2 -21548.13} C_VEL
LIN {X 0,Y 222.695,Z 432.51,A -85,B 0,C 180,E1 -21550.473,E2 -21550.473} C_VEL
LIN {X 0,Y 219.627,Z 420.765,A -85,B 0,C 180,E1 -21552.946,E2 -21552.946} C_VEL
LIN {X 0,Y 216.196,Z 411.904,A -85,B 0,C 180,E1 -21554.951,E2 -21554.951} C_VEL
LIN {X 0,Y 212.495,Z 404.474,A -85,B 0,C 180,E1 -21556.817,E2 -21556.817} C_VEL
LIN {X 0,Y 210.428,Z 400.751,A -85,B 0,C 180,E1 -21557.823,E2 -21557.823} C_VEL
LIN {X 0,Y 207.776,Z 396.347,A -85,B 0,C 180,E1 -21559.053,E2 -21559.053} C_VEL
LIN {X 0,Y 205.444,Z 392.617,A -85,B 0,C 180,E1 -21560.151,E2 -21560.151} C_VEL
LIN {X 0,Y 204.668,Z 391.48,A -85,B 0,C 180,E1 -21560.5,E2 -21560.5} C_VEL
LIN {X 0,Y 202.349,Z 388.574,A -85,B 0,C 180,E1 -21561.543,E2 -21561.543} C_VEL
LIN {X 0,Y 201.488,Z 386.267,A -85,B 0,C 180,E1 -21562.065,E2 -21562.065} C_VEL
LIN {X 0,Y 201.114,Z 383.798,A -85,B 0,C 180,E1 -21567.003,E2 -21567.003} C_VEL
LIN {X 0,Y 200.82,Z 382.038,A -85,B 0,C 180,E1 -21571.036,E2 -21571.036} C_VEL
LIN {X 0,Y 200.52,Z 380.328,A -85,B 0,C 180,E1 -21575.683,E2 -21575.683} C_VEL
LIN {X 0,Y 200.313,Z 378.608,A -85,B 0,C 180,E1 -21581.593,E2 -21581.593} C_VEL
LIN {X 0,Y 200.159,Z 377.78,A -85,B 0,C 180,E1 -21585.771,E2 -21585.771} C_VEL
LIN {X 0,Y 200.267,Z 377.147,A -85,B 0,C 180,E1 -21589.894,E2 -21589.894} C_VEL
LIN {X 0,Y 200.172,Z 376.873,A -85,B 0,C 180,E1 -21593.953,E2 -21593.953} C_VEL
LIN {X 0,Y 200.436,Z 376.801,A -85,B 0,C 180,E1 -21597.99,E2 -21597.99} C_VEL
LIN {X 0,Y 200.618,Z 376.896,A -85,B 0,C 180,E1 -21600,E2 -21600} C_VEL
LIN {X 0,Y 200.319,Z 377.477,A -85,B 0,C 180,E1 -21604.023,E2 -21604.023} C_VEL
LIN {X 0,Y 200.503,Z 378.224,A -85,B 0,C 180,E1 -21608.059,E2 -21608.059} C_VEL
LIN {X 0,Y 200.534,Z 379.351,A -85,B 0,C 180,E1 -21612.138,E2 -21612.138} C_VEL
LIN {X 0,Y 200.81,Z 380.78,A -85,B 0,C 180,E1 -21616.259,E2 -21616.259} C_VEL
LIN {X 0,Y 201.063,Z 382.569,A -85,B 0,C 180,E1 -21620.459,E2 -21620.459} C_VEL
LIN {X 0,Y 201.493,Z 384.823,A -85,B 0,C 180,E1 -21624.922,E2 -21624.922} C_VEL
LIN {X 0,Y 201.962,Z 387.554,A -85,B 0,C 180,E1 -21629.544,E2 -21629.544} C_VEL
LIN {X 0,Y 202.616,Z 391.212,A -85,B 0,C 180,E1 -21634.912,E2 -21634.912} C_VEL
LIN {X 0,Y 202.729,Z 391.88,A -85,B 0,C 180,E1 -21635.803,E2 -21635.803} C_VEL
LIN {X 0,Y 204.132,Z 395.088,A -85,B 0,C 180,E1 -21636.517,E2 -21636.517} C_VEL
LIN {X 0,Y 206.484,Z 398.029,A -85,B 0,C 180,E1 -21637.537,E2 -21637.537} C_VEL
LIN {X 0,Y 208.782,Z 402.14,A -85,B 0,C 180,E1 -21638.594,E2 -21638.594} C_VEL
LIN {X 0,Y 209.936,Z 403.914,A -85,B 0,C 180,E1 -21639.111,E2 -21639.111} C_VEL
LIN {X 0,Y 213.277,Z 410.143,A -85,B 0,C 180,E1 -21640.665,E2 -21640.665} C_VEL
LIN {X 0,Y 217.09,Z 417.62,A -85,B 0,C 180,E1 -21642.484,E2 -21642.484} C_VEL
LIN {X 0,Y 221.967,Z 429.473,A -85,B 0,C 180,E1 -21645.109,E2 -21645.109} C_VEL
LIN {X 0,Y 223.067,Z 433.143,A -85,B 0,C 180,E1 -21645.853,E2 -21645.853} C_VEL
LIN {X 0,Y 224.319,Z 445.589,A -85,B 0,C 180,E1 -21647.951,E2 -21647.951} C_VEL
LIN {X 0,Y 224.684,Z 458.528,A -85,B 0,C 180,E1 -21650.282,E2 -21650.282} C_VEL
LIN {X 0,Y 224.178,Z 467.736,A -85,B 0,C 180,E1 -21652.054,E2 -21652.054} C_VEL
LIN {X 0,Y 219.702,Z 480.591,A -85,B 0,C 180,E1 -21654.282,E2 -21654.282} C_VEL
LIN {X 0,Y 215.261,Z 492.294,A -85,B 0,C 180,E1 -21656.847,E2 -21656.847} C_VEL
LIN {X 0,Y 211.329,Z 502.094,A -85,B 0,C 180,E1 -21659.525,E2 -21659.525} C_VEL
LIN {X 0,Y 207.529,Z 511.68,A -85,B 0,C 180,E1 -21662.794,E2 -21662.794} C_VEL
LIN {X 0,Y 206.121,Z 514.99,A -85,B 0,C 180,E1 -21664.103,E2 -21664.103} C_VEL
LIN {X 0,Y 204.116,Z 518.15,A -85,B 0,C 180,E1 -21665.391,E2 -21665.391} C_VEL
LIN {X 0,Y 199.383,Z 522.872,A -85,B 0,C 180,E1 -21667.469,E2 -21667.469} C_VEL
LIN {X 0,Y 194.909,Z 527.115,A -85,B 0,C 180,E1 -21669.721,E2 -21669.721} C_VEL
LIN {X 0,Y 193.353,Z 529.426,A -85,B 0,C 180,E1 -21671.251,E2 -21671.251} C_VEL
LIN {X 0,Y 191.623,Z 534.2,A -85,B 0,C 180,E1 -21675.123,E2 -21675.123} C_VEL
LIN {X 0,Y 190.585,Z 538.057,A -85,B 0,C 180,E1 -21679.375,E2 -21679.375} C_VEL
LIN {X 0,Y 190.285,Z 540.609,A -85,B 0,C 180,E1 -21683.638,E2 -21683.638} C_VEL
LIN {X 0,Y 190.315,Z 541.41,A -85,B 0,C 180,E1 -21685.764,E2 -21685.764} C_VEL
LIN {X 0,Y 190.498,Z 542.062,A -85,B 0,C 180,E1 -21690,E2 -21690} C_VEL
LIN {X 0,Y 190.329,Z 541.341,A -85,B 0,C 180,E1 -21694.45,E2 -21694.45} C_VEL
LIN {X 0,Y 190.366,Z 539.459,A -85,B 0,C 180,E1 -21698.492,E2 -21698.492} C_VEL
LIN {X 0,Y 190.975,Z 536.246,A -85,B 0,C 180,E1 -21702.756,E2 -21702.756} C_VEL
LIN {X 0,Y 192.431,Z 531.698,A -85,B 0,C 180,E1 -21706.988,E2 -21706.988} C_VEL
LIN {X 0,Y 194.762,Z 525.7,A -85,B 0,C 180,E1 -21711.152,E2 -21711.152} C_VEL
LIN {X 0,Y 197.968,Z 518.097,A -85,B 0,C 180,E1 -21715.215,E2 -21715.215} C_VEL
LIN {X 0,Y 201.61,Z 509.919,A -85,B 0,C 180,E1 -21718.641,E2 -21718.641} C_VEL
LIN {X 0,Y 205.79,Z 500.05,A -85,B 0,C 180,E1 -21721.961,E2 -21721.961} C_VEL
LIN {X 0,Y 210.003,Z 489.909,A -85,B 0,C 180,E1 -21724.675,E2 -21724.675} C_VEL
LIN {X 0,Y 214.3,Z 478.877,A -85,B 0,C 180,E1 -21727.057,E2 -21727.057} C_VEL
LIN {X 0,Y 218.033,Z 468.553,A -85,B 0,C 180,E1 -21728.864,E2 -21728.864} C_VEL
LIN {X 0,Y 218.617,Z 457.415,A -85,B 0,C 180,E1 -21731.097,E2 -21731.097} C_VEL
LIN {X 0,Y 218.299,Z 444.294,A -85,B 0,C 180,E1 -21733.536,E2 -21733.536} C_VEL
LIN {X 0,Y 217.393,Z 435.395,A -85,B 0,C 180,E1 -21735.125,E2 -21735.125} C_VEL
LIN {X 0,Y 213.545,Z 424.834,A -85,B 0,C 180,E1 -21737.571,E2 -21737.571} C_VEL
LIN {X 0,Y 209.748,Z 416.462,A -85,B 0,C 180,E1 -21739.668,E2 -21739.668} C_VEL
LIN {X 0,Y 206.944,Z 410.981,A -85,B 0,C 180,E1 -21741.116,E2 -21741.116} C_VEL
LIN {X 0,Y 205.081,Z 407.488,A -85,B 0,C 180,E1 -21742.084,E2 -21742.084} C_VEL
LIN {X 0,Y 202.385,Z 402.836,A -85,B 0,C 180,E1 -21743.433,E2 -21743.433} C_VEL
LIN {X 0,Y 199.969,Z 399.125,A -85,B 0,C 180,E1 -21744.634,E2 -21744.634} C_VEL
LIN {X 0,Y 199.01,Z 397.309,A -85,B 0,C 180,E1 -21745.134,E2 -21745.134} C_VEL
LIN {X 0,Y 196.625,Z 394.372,A -85,B 0,C 180,E1 -21746.306,E2 -21746.306} C_VEL
LIN {X 0,Y 195.453,Z 391.585,A -85,B 0,C 180,E1 -21747.02,E2 -21747.02} C_VEL
LIN {X 0,Y 194.934,Z 388.375,A -85,B 0,C 180,E1 -21752.051,E2 -21752.051} C_VEL
LIN {X 0,Y 194.488,Z 385.929,A -85,B 0,C 180,E1 -21756.579,E2 -21756.579} C_VEL
LIN {X 0,Y 194.127,Z 383.863,A -85,B 0,C 180,E1 -21760.985,E2 -21760.985} C_VEL
LIN {X 0,Y 193.872,Z 382.194,A -85,B 0,C 180,E1 -21765.301,E2 -21765.301} C_VEL
LIN {X 0,Y 193.76,Z 380.832,A -85,B 0,C 180,E1 -21769.551,E2 -21769.551} C_VEL
LIN {X 0,Y 193.572,Z 379.888,A -85,B 0,C 180,E1 -21773.747,E2 -21773.747} C_VEL
LIN {X 0,Y 193.724,Z 379.161,A -85,B 0,C 180,E1 -21777.921,E2 -21777.921} C_VEL
LIN {X 0,Y 193.815,Z 378.913,A -85,B 0,C 180,E1 -21780,E2 -21780} C_VEL
LIN {X 0,Y 193.355,Z 378.871,A -85,B 0,C 180,E1 -21784.169,E2 -21784.169} C_VEL
LIN {X 0,Y 193.46,Z 378.959,A -85,B 0,C 180,E1 -21788.356,E2 -21788.356} C_VEL
LIN {X 0,Y 193.337,Z 379.436,A -85,B 0,C 180,E1 -21792.598,E2 -21792.598} C_VEL
LIN {X 0,Y 193.401,Z 380.191,A -85,B 0,C 180,E1 -21796.901,E2 -21796.901} C_VEL
LIN {X 0,Y 193.511,Z 381.257,A -85,B 0,C 180,E1 -21801.296,E2 -21801.296} C_VEL
LIN {X 0,Y 193.742,Z 382.653,A -85,B 0,C 180,E1 -21805.805,E2 -21805.805} C_VEL
LIN {X 0,Y 194.02,Z 384.438,A -85,B 0,C 180,E1 -21810.473,E2 -21810.473} C_VEL
LIN {X 0,Y 194.384,Z 386.543,A -85,B 0,C 180,E1 -21815.219,E2 -21815.219} C_VEL
LIN {X 0,Y 195.992,Z 389.888,A -85,B 0,C 180,E1 -21816.221,E2 -21816.221} C_VEL
LIN {X 0,Y 198.405,Z 392.694,A -85,B 0,C 180,E1 -21817.414,E2 -21817.414} C_VEL
LIN {X 0,Y 200.534,Z 396.285,A -85,B 0,C 180,E1 -21818.548,E2 -21818.548} C_VEL
LIN {X 0,Y 201.946,Z 398.16,A -85,B 0,C 180,E1 -21819.243,E2 -21819.243} C_VEL
LIN {X 0,Y 204.187,Z 401.899,A -85,B 0,C 180,E1 -21820.397,E2 -21820.397} C_VEL
LIN {X 0,Y 207.741,Z 408.301,A -85,B 0,C 180,E1 -21822.267,E2 -21822.267} C_VEL
LIN {X 0,Y 212.092,Z 417.678,A -85,B 0,C 180,E1 -21824.762,E2 -21824.762} C_VEL
LIN {X 0,Y 215.071,Z 426.808,A -85,B 0,C 180,E1 -21826.887,E2 -21826.887} C_VEL
LIN {X 0,Y 217.221,Z 436.573,A -85,B 0,C 180,E1 -21829.061,E2 -21829.061} C_VEL
LIN {X 0,Y 218.659,Z 447.369,A -85,B 0,C 180,E1 -21831.453,E2 -21831.453} C_VEL
LIN {X 0,Y 219.146,Z 456.859,A -85,B 0,C 180,E1 -21833.639,E2 -21833.639} C_VEL
LIN {X 0,Y 217.828,Z 461.505,A -85,B 0,C 180,E1 -21834.496,E2 -21834.496} C_VEL
LIN {X 0,Y 213.846,Z 472.081,A -85,B 0,C 180,E1 -21836.6,E2 -21836.6} C_VEL
LIN {X 0,Y 209.625,Z 482.614,A -85,B 0,C 180,E1 -21839.251,E2 -21839.251} C_VEL
LIN {X 0,Y 205.609,Z 491.369,A -85,B 0,C 180,E1 -21841.966,E2 -21841.966} C_VEL
LIN {X 0,Y 201.615,Z 499.796,A -85,B 0,C 180,E1 -21845.273,E2 -21845.273} C_VEL
LIN {X 0,Y 198.836,Z 505.75,A -85,B 0,C 180,E1 -21848.215,E2 -21848.215} C_VEL
LIN {X 0,Y 195.578,Z 512.139,A -85,B 0,C 180,E1 -21852.215,E2 -21852.215} C_VEL
LIN {X 0,Y 193.268,Z 516.964,A -85,B 0,C 180,E1 -21856.328,E2 -21856.328} C_VEL
LIN {X 0,Y 192.055,Z 519.688,A -85,B 0,C 180,E1 -21859.457,E2 -21859.457} C_VEL
LIN {X 0,Y 191.053,Z 522.135,A -85,B 0,C 180,E1 -21863.664,E2 -21863.664} C_VEL
LIN {X 0,Y 190.613,Z 523.351,A -85,B 0,C 180,E1 -21867.887,E2 -21867.887} C_VEL
LIN {X 0,Y 190.612,Z 523.37,A -85,B 0,C 180,E1 -21872.113,E2 -21872.113} C_VEL
LIN {X 0,Y 191.053,Z 522.195,A -85,B 0,C 180,E1 -21876.336,E2 -21876.336} C_VEL
LIN {X 0,Y 192.007,Z 519.791,A -85,B 0,C 180,E1 -21880.546,E2 -21880.546} C_VEL
LIN {X 0,Y 193.732,Z 516.074,A -85,B 0,C 180,E1 -21884.711,E2 -21884.711} C_VEL
LIN {X 0,Y 196.182,Z 510.939,A -85,B 0,C 180,E1 -21888.809,E2 -21888.809} C_VEL
LIN {X 0,Y 199.764,Z 504.159,A -85,B 0,C 180,E1 -21892.768,E2 -21892.768} C_VEL
LIN {X 0,Y 203.219,Z 496.659,A -85,B 0,C 180,E1 -21896.2,E2 -21896.2} C_VEL
LIN {X 0,Y 206.791,Z 489.051,A -85,B 0,C 180,E1 -21898.967,E2 -21898.967} C_VEL
LIN {X 0,Y 210.876,Z 479.83,A -85,B 0,C 180,E1 -21901.663,E2 -21901.663} C_VEL
LIN {X 0,Y 214.593,Z 470.658,A -85,B 0,C 180,E1 -21903.832,E2 -21903.832} C_VEL
LIN {X 0,Y 218.819,Z 458.973,A -85,B 0,C 180,E1 -21906.083,E2 -21906.083} C_VEL
LIN {X 0,Y 219.269,Z 456.957,A -85,B 0,C 180,E1 -21906.467,E2 -21906.467} C_VEL
LIN {X 0,Y 218.561,Z 445.424,A -85,B 0,C 180,E1 -21909.126,E2 -21909.126} C_VEL
LIN {X 0,Y 216.834,Z 434.217,A -85,B 0,C 180,E1 -21911.623,E2 -21911.623} C_VEL
LIN {X 0,Y 214.392,Z 424.196,A -85,B 0,C 180,E1 -21913.847,E2 -21913.847} C_VEL
LIN {X 0,Y 211.533,Z 416.327,A -85,B 0,C 180,E1 -21915.756,E2 -21915.756} C_VEL
LIN {X 0,Y 206.995,Z 406.705,A -85,B 0,C 180,E1 -21918.339,E2 -21918.339} C_VEL
LIN {X 0,Y 203.849,Z 401.434,A -85,B 0,C 180,E1 -21919.964,E2 -21919.964} C_VEL
LIN {X 0,Y 201.155,Z 396.998,A -85,B 0,C 180,E1 -21921.352,E2 -21921.352} C_VEL
LIN {X 0,Y 198.812,Z 393.551,A -85,B 0,C 180,E1 -21922.569,E2 -21922.569} C_VEL
LIN {X 0,Y 197.896,Z 391.929,A -85,B 0,C 180,E1 -21923.053,E2 -21923.053} C_VEL
LIN {X 0,Y 195.325,Z 388.906,A -85,B 0,C 180,E1 -21924.353,E2 -21924.353} C_VEL
LIN {X 0,Y 194.358,Z 386.548,A -85,B 0,C 180,E1 -21925.024,E2 -21925.024} C_VEL
LIN {X 0,Y 194.254,Z 385.576,A -85,B 0,C 180,E1 -21927.133,E2 -21927.133} C_VEL
LIN {X 0,Y 193.928,Z 383.587,A -85,B 0,C 180,E1 -21931.892,E2 -21931.892} C_VEL
LIN {X 0,Y 193.646,Z 382.03,A -85,B 0,C 180,E1 -21936.47,E2 -21936.47} C_VEL
LIN {X 0,Y 193.49,Z 380.803,A -85,B 0,C 180,E1 -21940.919,E2 -21940.919} C_VEL
LIN {X 0,Y 193.353,Z 379.921,A -85,B 0,C 180,E1 -21945.259,E2 -21945.259} C_VEL
LIN {X 0,Y 193.48,Z 379.315,A -85,B 0,C 180,E1 -21949.535,E2 -21949.535} C_VEL
LIN {X 0,Y 193.4,Z 379.014,A -85,B 0,C 180,E1 -21953.741,E2 -21953.741} C_VEL
LIN {X 0,Y 193.645,Z 378.938,A -85,B 0,C 180,E1 -21957.92,E2 -21957.92} C_VEL
LIN {X 0,Y 193.865,Z 379.021,A -85,B 0,C 180,E1 -21960,E2 -21960} C_VEL
LIN {X 0,Y 193.58,Z 379.668,A -85,B 0,C 180,E1 -21964.164,E2 -21964.164} C_VEL
LIN {X 0,Y 193.749,Z 380.439,A -85,B 0,C 180,E1 -21968.342,E2 -21968.342} C_VEL
LIN {X 0,Y 193.769,Z 381.598,A -85,B 0,C 180,E1 -21972.569,E2 -21972.569} C_VEL
LIN {X 0,Y 194.053,Z 383.067,A -85,B 0,C 180,E1 -21976.842,E2 -21976.842} C_VEL
LIN {X 0,Y 194.307,Z 384.951,A -85,B 0,C 180,E1 -21981.204,E2 -21981.204} C_VEL
LIN {X 0,Y 194.725,Z 387.182,A -85,B 0,C 180,E1 -21985.664,E2 -21985.664} C_VEL
LIN {X 0,Y 195.162,Z 389.882,A -85,B 0,C 180,E1 -21990.275,E2 -21990.275} C_VEL
LIN {X 0,Y 195.466,Z 391.609,A -85,B 0,C 180,E1 -21992.893,E2 -21992.893} C_VEL
LIN {X 0,Y 196.672,Z 394.482,A -85,B 0,C 180,E1 -21993.601,E2 -21993.601} C_VEL
LIN {X 0,Y 199.18,Z 397.481,A -85,B 0,C 180,E1 -21994.831,E2 -21994.831} C_VEL
LIN {X 0,Y 201.642,Z 401.869,A -85,B 0,C 180,E1 -21996.103,E2 -21996.103} C_VEL
LIN {X 0,Y 203.075,Z 403.939,A -85,B 0,C 180,E1 -21996.809,E2 -21996.809} C_VEL
LIN {X 0,Y 206.551,Z 410.217,A -85,B 0,C 180,E1 -21998.582,E2 -21998.582} C_VEL
LIN {X 0,Y 209.4,Z 415.725,A -85,B 0,C 180,E1 -22000.053,E2 -22000.053} C_VEL
LIN {X 0,Y 212.099,Z 421.298,A -85,B 0,C 180,E1 -22001.506,E2 -22001.506} C_VEL
LIN {X 0,Y 216.613,Z 432.803,A -85,B 0,C 180,E1 -22004.233,E2 -22004.233} C_VEL
LIN {X 0,Y 217.534,Z 435.819,A -85,B 0,C 180,E1 -22004.896,E2 -22004.896} C_VEL
LIN {X 0,Y 218.55,Z 447.867,A -85,B 0,C 180,E1 -22007.068,E2 -22007.068} C_VEL
LIN {X 0,Y 218.62,Z 460.897,A -85,B 0,C 180,E1 -22009.546,E2 -22009.546} C_VEL
LIN {X 0,Y 218.093,Z 468.719,A -85,B 0,C 180,E1 -22011.124,E2 -22011.124} C_VEL
LIN {X 0,Y 213.523,Z 481.254,A -85,B 0,C 180,E1 -22013.374,E2 -22013.374} C_VEL
LIN {X 0,Y 209.294,Z 491.902,A -85,B 0,C 180,E1 -22015.773,E2 -22015.773} C_VEL
LIN {X 0,Y 205.154,Z 501.716,A -85,B 0,C 180,E1 -22018.505,E2 -22018.505} C_VEL
LIN {X 0,Y 201.148,Z 511.312,A -85,B 0,C 180,E1 -22021.856,E2 -22021.856} C_VEL
LIN {X 0,Y 197.512,Z 519.241,A -85,B 0,C 180,E1 -22025.285,E2 -22025.285} C_VEL
LIN {X 0,Y 194.769,Z 525.787,A -85,B 0,C 180,E1 -22028.848,E2 -22028.848} C_VEL
LIN {X 0,Y 193.353,Z 529.426,A -85,B 0,C 180,E1 -22031.251,E2 -22031.251} C_VEL
LIN {X 0,Y 191.892,Z 531.588,A -85,B 0,C 180,E1 -22032.83,E2 -22032.83} C_VEL
LIN {X 0,Y 187.972,Z 534.62,A -85,B 0,C 180,E1 -22035.422,E2 -22035.422} C_VEL
LIN {X 0,Y 184.925,Z 536.654,A -85,B 0,C 180,E1 -22037.598,E2 -22037.598} C_VEL
LIN {X 0,Y 183.548,Z 537.974,A -85,B 0,C 180,E1 -22039.346,E2 -22039.346} C_VEL
LIN {X 0,Y 183.381,Z 538.348,A -85,B 0,C 180,E1 -22039.948,E2 -22039.948} C_VEL
LIN {X 0,Y 183.199,Z 540.263,A -85,B 0,C 180,E1 -22043.391,E2 -22043.391} C_VEL
LIN {X 0,Y 183.226,Z 541.104,A -85,B 0,C 180,E1 -22045.768,E2 -22045.768} C_VEL
LIN {X 0,Y 183.413,Z 541.717,A -85,B 0,C 180,E1 -22050,E2 -22050} C_VEL
LIN {X 0,Y 183.231,Z 541.05,A -85,B 0,C 180,E1 -22054.399,E2 -22054.399} C_VEL
LIN {X 0,Y 183.284,Z 539.11,A -85,B 0,C 180,E1 -22058.823,E2 -22058.823} C_VEL
LIN {X 0,Y 183.984,Z 535.896,A -85,B 0,C 180,E1 -22063.25,E2 -22063.25} C_VEL
LIN {X 0,Y 185.579,Z 531.346,A -85,B 0,C 180,E1 -22067.636,E2 -22067.636} C_VEL
LIN {X 0,Y 188.072,Z 525.343,A -85,B 0,C 180,E1 -22071.943,E2 -22071.943} C_VEL
LIN {X 0,Y 191.501,Z 517.736,A -85,B 0,C 180,E1 -22076.129,E2 -22076.129} C_VEL
LIN {X 0,Y 195.328,Z 509.549,A -85,B 0,C 180,E1 -22079.652,E2 -22079.652} C_VEL
LIN {X 0,Y 199.721,Z 499.668,A -85,B 0,C 180,E1 -22083.054,E2 -22083.054} C_VEL
LIN {X 0,Y 204.173,Z 489.514,A -85,B 0,C 180,E1 -22085.815,E2 -22085.815} C_VEL
LIN {X 0,Y 208.209,Z 479.533,A -85,B 0,C 180,E1 -22088.026,E2 -22088.026} C_VEL
LIN {X 0,Y 211.982,Z 469.546,A -85,B 0,C 180,E1 -22089.848,E2 -22089.848} C_VEL
LIN {X 0,Y 212.687,Z 458.774,A -85,B 0,C 180,E1 -22092.111,E2 -22092.111} C_VEL
LIN {X 0,Y 212.594,Z 446.461,A -85,B 0,C 180,E1 -22094.516,E2 -22094.516} C_VEL
LIN {X 0,Y 212.07,Z 439.154,A -85,B 0,C 180,E1 -22095.898,E2 -22095.898} C_VEL
LIN {X 0,Y 208.76,Z 429.267,A -85,B 0,C 180,E1 -22098.326,E2 -22098.326} C_VEL
LIN {X 0,Y 203.664,Z 417.506,A -85,B 0,C 180,E1 -22101.465,E2 -22101.465} C_VEL
LIN {X 0,Y 200.902,Z 412.299,A -85,B 0,C 180,E1 -22103.025,E2 -22103.025} C_VEL
LIN {X 0,Y 198.531,Z 407.95,A -85,B 0,C 180,E1 -22104.386,E2 -22104.386} C_VEL
LIN {X 0,Y 196.107,Z 403.735,A -85,B 0,C 180,E1 -22105.741,E2 -22105.741} C_VEL
LIN {X 0,Y 193.064,Z 399.203,A -85,B 0,C 180,E1 -22107.448,E2 -22107.448} C_VEL
LIN {X 0,Y 192.189,Z 397.401,A -85,B 0,C 180,E1 -22107.979,E2 -22107.979} C_VEL
LIN {X 0,Y 189.568,Z 394.406,A -85,B 0,C 180,E1 -22109.444,E2 -22109.444} C_VEL
LIN {X 0,Y 188.215,Z 391.246,A -85,B 0,C 180,E1 -22110.392,E2 -22110.392} C_VEL
LIN {X 0,Y 187.737,Z 388.343,A -85,B 0,C 180,E1 -22115.683,E2 -22115.683} C_VEL
LIN {X 0,Y 187.359,Z 386.22,A -85,B 0,C 180,E1 -22120.27,E2 -22120.27} C_VEL
LIN {X 0,Y 187.109,Z 384.464,A -85,B 0,C 180,E1 -22124.757,E2 -22124.757} C_VEL
LIN {X 0,Y 186.96,Z 383.065,A -85,B 0,C 180,E1 -22129.167,E2 -22129.167} C_VEL
LIN {X 0,Y 186.801,Z 382.03,A -85,B 0,C 180,E1 -22133.52,E2 -22133.52} C_VEL
LIN {X 0,Y 186.937,Z 381.299,A -85,B 0,C 180,E1 -22137.846,E2 -22137.846} C_VEL
LIN {X 0,Y 187.054,Z 381.043,A -85,B 0,C 180,E1 -22140,E2 -22140} C_VEL
LIN {X 0,Y 186.579,Z 380.982,A -85,B 0,C 180,E1 -22144.321,E2 -22144.321} C_VEL
LIN {X 0,Y 186.662,Z 381.065,A -85,B 0,C 180,E1 -22148.662,E2 -22148.662} C_VEL
LIN {X 0,Y 186.522,Z 381.566,A -85,B 0,C 180,E1 -22153.067,E2 -22153.067} C_VEL
LIN {X 0,Y 186.593,Z 382.363,A -85,B 0,C 180,E1 -22157.537,E2 -22157.537} C_VEL
LIN {X 0,Y 186.708,Z 383.482,A -85,B 0,C 180,E1 -22162.112,E2 -22162.112} C_VEL
LIN {X 0,Y 186.948,Z 384.943,A -85,B 0,C 180,E1 -22166.816,E2 -22166.816} C_VEL
LIN {X 0,Y 187.187,Z 386.234,A -85,B 0,C 180,E1 -22170.283,E2 -22170.283} C_VEL
LIN {X 0,Y 187.302,Z 387.058,A -85,B 0,C 180,E1 -22171.927,E2 -22171.927} C_VEL
LIN {X 0,Y 188.661,Z 389.857,A -85,B 0,C 180,E1 -22172.853,E2 -22172.853} C_VEL
LIN {X 0,Y 191.238,Z 392.565,A -85,B 0,C 180,E1 -22174.316,E2 -22174.316} C_VEL
LIN {X 0,Y 193.865,Z 396.872,A -85,B 0,C 180,E1 -22175.898,E2 -22175.898} C_VEL
LIN {X 0,Y 195.176,Z 398.528,A -85,B 0,C 180,E1 -22176.62,E2 -22176.62} C_VEL
LIN {X 0,Y 197.586,Z 402.487,A -85,B 0,C 180,E1 -22178.01,E2 -22178.01} C_VEL
LIN {X 0,Y 201.37,Z 409.212,A -85,B 0,C 180,E1 -22180.215,E2 -22180.215} C_VEL
LIN {X 0,Y 204.578,Z 415.422,A -85,B 0,C 180,E1 -22182.123,E2 -22182.123} C_VEL
LIN {X 0,Y 208.123,Z 424.325,A -85,B 0,C 180,E1 -22184.552,E2 -22184.552} C_VEL
LIN {X 0,Y 210.571,Z 433.613,A -85,B 0,C 180,E1 -22186.795,E2 -22186.795} C_VEL
LIN {X 0,Y 212.225,Z 444.074,A -85,B 0,C 180,E1 -22189.247,E2 -22189.247} C_VEL
LIN {X 0,Y 213.033,Z 454.558,A -85,B 0,C 180,E1 -22191.754,E2 -22191.754} C_VEL
LIN {X 0,Y 213.047,Z 458.995,A -85,B 0,C 180,E1 -22192.829,E2 -22192.829} C_VEL
LIN {X 0,Y 209.255,Z 469.561,A -85,B 0,C 180,E1 -22194.889,E2 -22194.889} C_VEL
LIN {X 0,Y 204.946,Z 479.76,A -85,B 0,C 180,E1 -22197.31,E2 -22197.31} C_VEL
LIN {X 0,Y 200.709,Z 489.035,A -85,B 0,C 180,E1 -22200.068,E2 -22200.068} C_VEL
LIN {X 0,Y 196.745,Z 497.129,A -85,B 0,C 180,E1 -22203.077,E2 -22203.077} C_VEL
LIN {X 0,Y 193.256,Z 504.242,A -85,B 0,C 180,E1 -22206.42,E2 -22206.42} C_VEL
LIN {X 0,Y 189.531,Z 511.082,A -85,B 0,C 180,E1 -22210.505,E2 -22210.505} C_VEL
LIN {X 0,Y 186.904,Z 516.279,A -85,B 0,C 180,E1 -22214.739,E2 -22214.739} C_VEL
LIN {X 0,Y 185.065,Z 520.035,A -85,B 0,C 180,E1 -22219.054,E2 -22219.054} C_VEL
LIN {X 0,Y 184.01,Z 522.481,A -85,B 0,C 180,E1 -22223.421,E2 -22223.421} C_VEL
LIN {X 0,Y 183.535,Z 523.696,A -85,B 0,C 180,E1 -22227.806,E2 -22227.806} C_VEL
LIN {X 0,Y 183.534,Z 523.714,A -85,B 0,C 180,E1 -22232.195,E2 -22232.195} C_VEL
LIN {X 0,Y 184.036,Z 522.443,A -85,B 0,C 180,E1 -22236.832,E2 -22236.832} C_VEL
LIN {X 0,Y 185.019,Z 520.136,A -85,B 0,C 180,E1 -22240.949,E2 -22240.949} C_VEL
LIN {X 0,Y 186.867,Z 516.42,A -85,B 0,C 180,E1 -22245.264,E2 -22245.264} C_VEL
LIN {X 0,Y 189.463,Z 511.288,A -85,B 0,C 180,E1 -22249.503,E2 -22249.503} C_VEL
LIN {X 0,Y 192.212,Z 506.349,A -85,B 0,C 180,E1 -22252.577,E2 -22252.577} C_VEL
LIN {X 0,Y 195.126,Z 500.459,A -85,B 0,C 180,E1 -22255.609,E2 -22255.609} C_VEL
LIN {X 0,Y 199.279,Z 492.1,A -85,B 0,C 180,E1 -22259.008,E2 -22259.008} C_VEL
LIN {X 0,Y 203.485,Z 483.429,A -85,B 0,C 180,E1 -22261.784,E2 -22261.784} C_VEL
LIN {X 0,Y 207.901,Z 472.997,A -85,B 0,C 180,E1 -22264.488,E2 -22264.488} C_VEL
LIN {X 0,Y 212.021,Z 462.548,A -85,B 0,C 180,E1 -22266.632,E2 -22266.632} C_VEL
LIN {X 0,Y 213.127,Z 459.397,A -85,B 0,C 180,E1 -22267.206,E2 -22267.206} C_VEL
LIN {X 0,Y 212.832,Z 449.221,A -85,B 0,C 180,E1 -22269.673,E2 -22269.673} C_VEL
LIN {X 0,Y 211.748,Z 439.709,A -85,B 0,C 180,E1 -22271.926,E2 -22271.926} C_VEL
LIN {X 0,Y 209.433,Z 428.476,A -85,B 0,C 180,E1 -22274.581,E2 -22274.581} C_VEL
LIN {X 0,Y 206.91,Z 420.857,A -85,B 0,C 180,E1 -22276.542,E2 -22276.542} C_VEL
LIN {X 0,Y 202.7,Z 411.558,A -85,B 0,C 180,E1 -22279.205,E2 -22279.205} C_VEL
LIN {X 0,Y 199.524,Z 405.883,A -85,B 0,C 180,E1 -22281.058,E2 -22281.058} C_VEL
LIN {X 0,Y 197.637,Z 402.591,A -85,B 0,C 180,E1 -22282.163,E2 -22282.163} C_VEL
LIN {X 0,Y 195.133,Z 398.453,A -85,B 0,C 180,E1 -22283.619,E2 -22283.619} C_VEL
LIN {X 0,Y 191.965,Z 393.96,A -85,B 0,C 180,E1 -22285.462,E2 -22285.462} C_VEL
LIN {X 0,Y 191.109,Z 392.463,A -85,B 0,C 180,E1 -22285.98,E2 -22285.98} C_VEL
LIN {X 0,Y 188.559,Z 389.754,A -85,B 0,C 180,E1 -22287.444,E2 -22287.444} C_VEL
LIN {X 0,Y 187.269,Z 386.882,A -85,B 0,C 180,E1 -22288.417,E2 -22288.417} C_VEL
LIN {X 0,Y 186.968,Z 385.05,A -85,B 0,C 180,E1 -22293.187,E2 -22293.187} C_VEL
LIN {X 0,Y 186.874,Z 384.26,A -85,B 0,C 180,E1 -22295.563,E2 -22295.563} C_VEL
LIN {X 0,Y 186.674,Z 382.981,A -85,B 0,C 180,E1 -22300.258,E2 -22300.258} C_VEL
LIN {X 0,Y 186.556,Z 382.065,A -85,B 0,C 180,E1 -22304.709,E2 -22304.709} C_VEL
LIN {X 0,Y 186.672,Z 381.429,A -85,B 0,C 180,E1 -22309.149,E2 -22309.149} C_VEL
LIN {X 0,Y 186.647,Z 381.15,A -85,B 0,C 180,E1 -22313.514,E2 -22313.514} C_VEL
LIN {X 0,Y 186.866,Z 381.071,A -85,B 0,C 180,E1 -22317.844,E2 -22317.844} C_VEL
LIN {X 0,Y 187.095,Z 381.149,A -85,B 0,C 180,E1 -22320,E2 -22320} C_VEL
LIN {X 0,Y 186.802,Z 381.805,A -85,B 0,C 180,E1 -22324.315,E2 -22324.315} C_VEL
LIN {X 0,Y 186.968,Z 382.651,A -85,B 0,C 180,E1 -22328.647,E2 -22328.647} C_VEL
LIN {X 0,Y 187.006,Z 383.848,A -85,B 0,C 180,E1 -22333.031,E2 -22333.031} C_VEL
LIN {X 0,Y 187.265,Z 385.372,A -85,B 0,C 180,E1 -22337.472,E2 -22337.472} C_VEL
LIN {X 0,Y 187.545,Z 387.317,A -85,B 0,C 180,E1 -22342.008,E2 -22342.008} C_VEL
LIN {X 0,Y 187.944,Z 389.652,A -85,B 0,C 180,E1 -22346.662,E2 -22346.662} C_VEL
LIN {X 0,Y 188.288,Z 391.484,A -85,B 0,C 180,E1 -22349.548,E2 -22349.548} C_VEL
LIN {X 0,Y 189.749,Z 394.676,A -85,B 0,C 180,E1 -22350.525,E2 -22350.525} C_VEL
LIN {X 0,Y 192.457,Z 397.886,A -85,B 0,C 180,E1 -22352.048,E2 -22352.048} C_VEL
LIN {X 0,Y 194.736,Z 401.89,A -85,B 0,C 180,E1 -22353.392,E2 -22353.392} C_VEL
LIN {X 0,Y 196.154,Z 403.774,A -85,B 0,C 180,E1 -22354.164,E2 -22354.164} C_VEL
LIN {X 0,Y 198.689,Z 408.113,A -85,B 0,C 180,E1 -22355.581,E2 -22355.581} C_VEL
LIN {X 0,Y 202.637,Z 415.527,A -85,B 0,C 180,E1 -22357.839,E2 -22357.839} C_VEL
LIN {X 0,Y 205.955,Z 422.293,A -85,B 0,C 180,E1 -22359.778,E2 -22359.778} C_VEL
LIN {X 0,Y 210.346,Z 433.58,A -85,B 0,C 180,E1 -22362.687,E2 -22362.687} C_VEL
LIN {X 0,Y 212.163,Z 439.331,A -85,B 0,C 180,E1 -22364.077,E2 -22364.077} C_VEL
LIN {X 0,Y 212.826,Z 449.915,A -85,B 0,C 180,E1 -22366.094,E2 -22366.094} C_VEL
LIN {X 0,Y 212.626,Z 462.532,A -85,B 0,C 180,E1 -22368.618,E2 -22368.618} C_VEL
LIN {X 0,Y 212.075,Z 469.676,A -85,B 0,C 180,E1 -22370.137,E2 -22370.137} C_VEL
LIN {X 0,Y 207.394,Z 481.916,A -85,B 0,C 180,E1 -22372.412,E2 -22372.412} C_VEL
LIN {X 0,Y 202.64,Z 493.31,A -85,B 0,C 180,E1 -22375.092,E2 -22375.092} C_VEL
LIN {X 0,Y 198.399,Z 502.846,A -85,B 0,C 180,E1 -22377.903,E2 -22377.903} C_VEL
LIN {X 0,Y 194.278,Z 512.2,A -85,B 0,C 180,E1 -22381.359,E2 -22381.359} C_VEL
LIN {X 0,Y 190.548,Z 519.915,A -85,B 0,C 180,E1 -22384.902,E2 -22384.902} C_VEL
LIN {X 0,Y 187.384,Z 527.092,A -85,B 0,C 180,E1 -22389.126,E2 -22389.126} C_VEL
LIN {X 0,Y 185.111,Z 532.695,A -85,B 0,C 180,E1 -22393.456,E2 -22393.456} C_VEL
LIN {X 0,Y 183.986,Z 535.944,A -85,B 0,C 180,E1 -22396.75,E2 -22396.75} C_VEL
LIN {X 0,Y 183.381,Z 538.348,A -85,B 0,C 180,E1 -22399.948,E2 -22399.948} C_VEL
LIN {X 0,Y 182.529,Z 539.448,A -85,B 0,C 180,E1 -22401.75,E2 -22401.75} C_VEL
LIN {X 0,Y 179.546,Z 540.638,A -85,B 0,C 180,E1 -22404.724,E2 -22404.724} C_VEL
LIN {X 0,Y 177.191,Z 541.159,A -85,B 0,C 180,E1 -22407.18,E2 -22407.18} C_VEL
LIN {X 0,Y 176.308,Z 541.315,A -85,B 0,C 180,E1 -22409.094,E2 -22409.094} C_VEL
LIN {X 0,Y 176.297,Z 541.353,A -85,B 0,C 180,E1 -22409.741,E2 -22409.741} C_VEL
LIN {X 0,Y 176.146,Z 540.815,A -85,B 0,C 180,E1 -22414.082,E2 -22414.082} C_VEL
LIN {X 0,Y 176.116,Z 539.89,A -85,B 0,C 180,E1 -22416.876,E2 -22416.876} C_VEL
LIN {X 0,Y 176.506,Z 537.315,A -85,B 0,C 180,E1 -22421.483,E2 -22421.483} C_VEL
LIN {X 0,Y 177.784,Z 533.443,A -85,B 0,C 180,E1 -22426.064,E2 -22426.064} C_VEL
LIN {X 0,Y 179.921,Z 528.177,A -85,B 0,C 180,E1 -22430.582,E2 -22430.582} C_VEL
LIN {X 0,Y 183.103,Z 521.392,A -85,B 0,C 180,E1 -22434.974,E2 -22434.974} C_VEL
LIN {X 0,Y 186.798,Z 514.042,A -85,B 0,C 180,E1 -22438.666,E2 -22438.666} C_VEL
LIN {X 0,Y 191.268,Z 504.575,A -85,B 0,C 180,E1 -22442.456,E2 -22442.456} C_VEL
LIN {X 0,Y 195.993,Z 494.416,A -85,B 0,C 180,E1 -22445.641,E2 -22445.641} C_VEL
LIN {X 0,Y 200.827,Z 483.319,A -85,B 0,C 180,E1 -22448.401,E2 -22448.401} C_VEL
LIN {X 0,Y 205.978,Z 470.553,A -85,B 0,C 180,E1 -22450.886,E2 -22450.886} C_VEL
LIN {X 0,Y 206.881,Z 459.053,A -85,B 0,C 180,E1 -22453.399,E2 -22453.399} C_VEL
LIN {X 0,Y 206.914,Z 446.983,A -85,B 0,C 180,E1 -22455.868,E2 -22455.868} C_VEL
LIN {X 0,Y 206.362,Z 441.276,A -85,B 0,C 180,E1 -22457.068,E2 -22457.068} C_VEL
LIN {X 0,Y 202.597,Z 430.041,A -85,B 0,C 180,E1 -22460.076,E2 -22460.076} C_VEL
LIN {X 0,Y 197.514,Z 418.392,A -85,B 0,C 180,E1 -22463.496,E2 -22463.496} C_VEL
LIN {X 0,Y 194.593,Z 413.053,A -85,B 0,C 180,E1 -22465.317,E2 -22465.317} C_VEL
LIN {X 0,Y 191.927,Z 408.181,A -85,B 0,C 180,E1 -22467.028,E2 -22467.028} C_VEL
LIN {X 0,Y 189.461,Z 404.028,A -85,B 0,C 180,E1 -22468.588,E2 -22468.588} C_VEL
LIN {X 0,Y 188.65,Z 402.828,A -85,B 0,C 180,E1 -22469.1,E2 -22469.1} C_VEL
LIN {X 0,Y 186.303,Z 399.404,A -85,B 0,C 180,E1 -22470.633,E2 -22470.633} C_VEL
LIN {X 0,Y 185.245,Z 397.236,A -85,B 0,C 180,E1 -22471.382,E2 -22471.382} C_VEL
LIN {X 0,Y 182.585,Z 394.382,A -85,B 0,C 180,E1 -22473.127,E2 -22473.127} C_VEL
LIN {X 0,Y 181.101,Z 391.246,A -85,B 0,C 180,E1 -22474.306,E2 -22474.306} C_VEL
LIN {X 0,Y 180.984,Z 390.776,A -85,B 0,C 180,E1 -22474.713,E2 -22474.713} C_VEL
LIN {X 0,Y 180.595,Z 388.576,A -85,B 0,C 180,E1 -22479.498,E2 -22479.498} C_VEL
LIN {X 0,Y 180.338,Z 386.746,A -85,B 0,C 180,E1 -22484.17,E2 -22484.17} C_VEL
LIN {X 0,Y 180.183,Z 385.3,A -85,B 0,C 180,E1 -22488.754,E2 -22488.754} C_VEL
LIN {X 0,Y 180.062,Z 384.226,A -85,B 0,C 180,E1 -22493.276,E2 -22493.276} C_VEL
LIN {X 0,Y 180.143,Z 383.446,A -85,B 0,C 180,E1 -22497.765,E2 -22497.765} C_VEL
LIN {X 0,Y 180.275,Z 383.174,A -85,B 0,C 180,E1 -22500,E2 -22500} C_VEL
LIN {X 0,Y 179.799,Z 383.12,A -85,B 0,C 180,E1 -22504.484,E2 -22504.484} C_VEL
LIN {X 0,Y 179.879,Z 383.223,A -85,B 0,C 180,E1 -22508.992,E2 -22508.992} C_VEL
LIN {X 0,Y 179.742,Z 383.744,A -85,B 0,C 180,E1 -22513.569,E2 -22513.569} C_VEL
LIN {X 0,Y 179.79,Z 384.57,A -85,B 0,C 180,E1 -22518.224,E2 -22518.224} C_VEL
LIN {X 0,Y 179.913,Z 385.704,A -85,B 0,C 180,E1 -22522.994,E2 -22522.994} C_VEL
LIN {X 0,Y 180.19,Z 387.3,A -85,B 0,C 180,E1 -22527.839,E2 -22527.839} C_VEL
LIN {X 0,Y 181.433,Z 390.002,A -85,B 0,C 180,E1 -22528.881,E2 -22528.881} C_VEL
LIN {X 0,Y 184.268,Z 392.978,A -85,B 0,C 180,E1 -22530.814,E2 -22530.814} C_VEL
LIN {X 0,Y 185.04,Z 394.207,A -85,B 0,C 180,E1 -22531.349,E2 -22531.349} C_VEL
LIN {X 0,Y 187.363,Z 397.67,A -85,B 0,C 180,E1 -22532.95,E2 -22532.95} C_VEL
LIN {X 0,Y 188.633,Z 399.133,A -85,B 0,C 180,E1 -22533.737,E2 -22533.737} C_VEL
LIN {X 0,Y 191.041,Z 403.116,A -85,B 0,C 180,E1 -22535.329,E2 -22535.329} C_VEL
LIN {X 0,Y 194.951,Z 409.807,A -85,B 0,C 180,E1 -22537.857,E2 -22537.857} C_VEL
LIN {X 0,Y 196.952,Z 413.473,A -85,B 0,C 180,E1 -22539.151,E2 -22539.151} C_VEL
LIN {X 0,Y 200.682,Z 421.519,A -85,B 0,C 180,E1 -22541.713,E2 -22541.713} C_VEL
LIN {X 0,Y 203.255,Z 428.585,A -85,B 0,C 180,E1 -22543.753,E2 -22543.753} C_VEL
LIN {X 0,Y 205.441,Z 438.425,A -85,B 0,C 180,E1 -22546.276,E2 -22546.276} C_VEL
LIN {X 0,Y 206.678,Z 448.327,A -85,B 0,C 180,E1 -22548.736,E2 -22548.736} C_VEL
LIN {X 0,Y 207.118,Z 458.431,A -85,B 0,C 180,E1 -22551.302,E2 -22551.302} C_VEL
LIN {X 0,Y 207.05,Z 460.39,A -85,B 0,C 180,E1 -22551.815,E2 -22551.815} C_VEL
LIN {X 0,Y 203.508,Z 469.969,A -85,B 0,C 180,E1 -22553.744,E2 -22553.744} C_VEL
LIN {X 0,Y 199.023,Z 480.15,A -85,B 0,C 180,E1 -22556.208,E2 -22556.208} C_VEL
LIN {X 0,Y 194.6,Z 489.411,A -85,B 0,C 180,E1 -22559.027,E2 -22559.027} C_VEL
LIN {X 0,Y 190.018,Z 498.326,A -85,B 0,C 180,E1 -22562.464,E2 -22562.464} C_VEL
LIN {X 0,Y 186.773,Z 504.6,A -85,B 0,C 180,E1 -22565.549,E2 -22565.549} C_VEL
LIN {X 0,Y 182.842,Z 511.435,A -85,B 0,C 180,E1 -22569.761,E2 -22569.761} C_VEL
LIN {X 0,Y 180.063,Z 516.627,A -85,B 0,C 180,E1 -22574.144,E2 -22574.144} C_VEL
LIN {X 0,Y 178.088,Z 520.382,A -85,B 0,C 180,E1 -22578.62,E2 -22578.62} C_VEL
LIN {X 0,Y 176.962,Z 522.826,A -85,B 0,C 180,E1 -22583.157,E2 -22583.157} C_VEL
LIN {X 0,Y 176.459,Z 524.041,A -85,B 0,C 180,E1 -22587.718,E2 -22587.718} C_VEL
LIN {X 0,Y 176.458,Z 524.059,A -85,B 0,C 180,E1 -22592.283,E2 -22592.283} C_VEL
LIN {X 0,Y 176.962,Z 522.884,A -85,B 0,C 180,E1 -22596.843,E2 -22596.843} C_VEL
LIN {X 0,Y 178.051,Z 520.481,A -85,B 0,C 180,E1 -22601.383,E2 -22601.383} C_VEL
LIN {X 0,Y 180.027,Z 516.766,A -85,B 0,C 180,E1 -22605.859,E2 -22605.859} C_VEL
LIN {X 0,Y 182.776,Z 511.637,A -85,B 0,C 180,E1 -22610.247,E2 -22610.247} C_VEL
LIN {X 0,Y 185.678,Z 506.699,A -85,B 0,C 180,E1 -22613.418,E2 -22613.418} C_VEL
LIN {X 0,Y 189.133,Z 500.053,A -85,B 0,C 180,E1 -22616.897,E2 -22616.897} C_VEL
LIN {X 0,Y 193.094,Z 492.466,A -85,B 0,C 180,E1 -22620.031,E2 -22620.031} C_VEL
LIN {X 0,Y 197.487,Z 483.808,A -85,B 0,C 180,E1 -22622.868,E2 -22622.868} C_VEL
LIN {X 0,Y 202.114,Z 473.393,A -85,B 0,C 180,E1 -22625.623,E2 -22625.623} C_VEL
LIN {X 0,Y 206.376,Z 462.971,A -85,B 0,C 180,E1 -22627.806,E2 -22627.806} C_VEL
LIN {X 0,Y 207.122,Z 460.83,A -85,B 0,C 180,E1 -22628.211,E2 -22628.211} C_VEL
LIN {X 0,Y 206.908,Z 449.784,A -85,B 0,C 180,E1 -22631.034,E2 -22631.034} C_VEL
LIN {X 0,Y 205.588,Z 438.897,A -85,B 0,C 180,E1 -22633.767,E2 -22633.767} C_VEL
LIN {X 0,Y 203.814,Z 430.522,A -85,B 0,C 180,E1 -22635.899,E2 -22635.899} C_VEL
LIN {X 0,Y 201.617,Z 423.724,A -85,B 0,C 180,E1 -22637.786,E2 -22637.786} C_VEL
LIN {X 0,Y 198.054,Z 415.762,A -85,B 0,C 180,E1 -22640.302,E2 -22640.302} C_VEL
LIN {X 0,Y 194.26,Z 408.365,A -85,B 0,C 180,E1 -22642.839,E2 -22642.839} C_VEL
LIN {X 0,Y 191.7,Z 403.964,A -85,B 0,C 180,E1 -22644.489,E2 -22644.489} C_VEL
LIN {X 0,Y 188.879,Z 399.708,A -85,B 0,C 180,E1 -22646.313,E2 -22646.313} C_VEL
LIN {X 0,Y 188.045,Z 398.383,A -85,B 0,C 180,E1 -22646.866,E2 -22646.866} C_VEL
LIN {X 0,Y 185.361,Z 394.821,A -85,B 0,C 180,E1 -22648.662,E2 -22648.662} C_VEL
LIN {X 0,Y 184.424,Z 393.06,A -85,B 0,C 180,E1 -22649.345,E2 -22649.345} C_VEL
LIN {X 0,Y 181.637,Z 390.318,A -85,B 0,C 180,E1 -22651.233,E2 -22651.233} C_VEL
LIN {X 0,Y 180.262,Z 387.543,A -85,B 0,C 180,E1 -22652.375,E2 -22652.375} C_VEL
LIN {X 0,Y 180.149,Z 387.174,A -85,B 0,C 180,E1 -22652.627,E2 -22652.627} C_VEL
LIN {X 0,Y 179.921,Z 385.818,A -85,B 0,C 180,E1 -22657.007,E2 -22657.007} C_VEL
LIN {X 0,Y 179.817,Z 384.666,A -85,B 0,C 180,E1 -22661.779,E2 -22661.779} C_VEL
LIN {X 0,Y 179.81,Z 383.668,A -85,B 0,C 180,E1 -22667.729,E2 -22667.729} C_VEL
LIN {X 0,Y 179.899,Z 383.346,A -85,B 0,C 180,E1 -22671.009,E2 -22671.009} C_VEL
LIN {X 0,Y 180.07,Z 383.209,A -85,B 0,C 180,E1 -22677.763,E2 -22677.763} C_VEL
LIN {X 0,Y 180.315,Z 383.281,A -85,B 0,C 180,E1 -22680,E2 -22680} C_VEL
LIN {X 0,Y 180.029,Z 383.94,A -85,B 0,C 180,E1 -22684.478,E2 -22684.478} C_VEL
LIN {X 0,Y 180.166,Z 384.815,A -85,B 0,C 180,E1 -22688.976,E2 -22688.976} C_VEL
LIN {X 0,Y 180.246,Z 386.068,A -85,B 0,C 180,E1 -22693.529,E2 -22693.529} C_VEL
LIN {X 0,Y 180.49,Z 387.692,A -85,B 0,C 180,E1 -22698.15,E2 -22698.15} C_VEL
LIN {X 0,Y 180.774,Z 389.712,A -85,B 0,C 180,E1 -22702.878,E2 -22702.878} C_VEL
LIN {X 0,Y 181.006,Z 390.944,A -85,B 0,C 180,E1 -22705.426,E2 -22705.426} C_VEL
LIN {X 0,Y 182.564,Z 394.353,A -85,B 0,C 180,E1 -22706.687,E2 -22706.687} C_VEL
LIN {X 0,Y 185.519,Z 397.692,A -85,B 0,C 180,E1 -22708.65,E2 -22708.65} C_VEL
LIN {X 0,Y 187.65,Z 401.631,A -85,B 0,C 180,E1 -22710.139,E2 -22710.139} C_VEL
LIN {X 0,Y 189.482,Z 403.998,A -85,B 0,C 180,E1 -22711.283,E2 -22711.283} C_VEL
LIN {X 0,Y 191.7,Z 407.852,A -85,B 0,C 180,E1 -22712.705,E2 -22712.705} C_VEL
LIN {X 0,Y 192.952,Z 409.933,A -85,B 0,C 180,E1 -22713.507,E2 -22713.507} C_VEL
LIN {X 0,Y 196.078,Z 415.693,A -85,B 0,C 180,E1 -22715.481,E2 -22715.481} C_VEL
LIN {X 0,Y 198.714,Z 421.067,A -85,B 0,C 180,E1 -22717.197,E2 -22717.197} C_VEL
LIN {X 0,Y 203.155,Z 431.471,A -85,B 0,C 180,E1 -22720.242,E2 -22720.242} C_VEL
LIN {X 0,Y 206.464,Z 441.448,A -85,B 0,C 180,E1 -22722.906,E2 -22722.906} C_VEL
LIN {X 0,Y 206.916,Z 444.496,A -85,B 0,C 180,E1 -22723.569,E2 -22723.569} C_VEL
LIN {X 0,Y 207.034,Z 456.345,A -85,B 0,C 180,E1 -22725.971,E2 -22725.971} C_VEL
LIN {X 0,Y 206.327,Z 468.162,A -85,B 0,C 180,E1 -22728.536,E2 -22728.536} C_VEL
LIN {X 0,Y 206.094,Z 470.67,A -85,B 0,C 180,E1 -22729.1,E2 -22729.1} C_VEL
LIN {X 0,Y 201.337,Z 482.556,A -85,B 0,C 180,E1 -22731.394,E2 -22731.394} C_VEL
LIN {X 0,Y 196.026,Z 494.603,A -85,B 0,C 180,E1 -22734.366,E2 -22734.366} C_VEL
LIN {X 0,Y 191.281,Z 504.765,A -85,B 0,C 180,E1 -22737.562,E2 -22737.562} C_VEL
LIN {X 0,Y 187.421,Z 513.035,A -85,B 0,C 180,E1 -22740.824,E2 -22740.824} C_VEL
LIN {X 0,Y 184.055,Z 519.555,A -85,B 0,C 180,E1 -22743.952,E2 -22743.952} C_VEL
LIN {X 0,Y 180.687,Z 526.737,A -85,B 0,C 180,E1 -22748.314,E2 -22748.314} C_VEL
LIN {X 0,Y 178.235,Z 532.344,A -85,B 0,C 180,E1 -22752.798,E2 -22752.798} C_VEL
LIN {X 0,Y 177.01,Z 535.595,A -85,B 0,C 180,E1 -22756.218,E2 -22756.218} C_VEL
LIN {X 0,Y 176.209,Z 538.797,A -85,B 0,C 180,E1 -22760.82,E2 -22760.82} C_VEL
LIN {X 0,Y 176.122,Z 540.718,A -85,B 0,C 180,E1 -22765.422,E2 -22765.422} C_VEL
LIN {X 0,Y 176.297,Z 541.353,A -85,B 0,C 180,E1 -22769.741,E2 -22769.741} C_VEL
LIN {X 0,Y 176.077,Z 541.372,A -85,B 0,C 180,E1 -22771.013,E2 -22771.013} C_VEL
LIN {X 0,Y 175.282,Z 541.254,A -85,B 0,C 180,E1 -22772.269,E2 -22772.269} C_VEL
LIN {X 0,Y 172.77,Z 540.66,A -85,B 0,C 180,E1 -22774.745,E2 -22774.745} C_VEL
LIN {X 0,Y 170.216,Z 539.623,A -85,B 0,C 180,E1 -22777.285,E2 -22777.285} C_VEL
LIN {X 0,Y 169.211,Z 538.588,A -85,B 0,C 180,E1 -22779.258,E2 -22779.258} C_VEL
LIN {X 0,Y 169.184,Z 538.197,A -85,B 0,C 180,E1 -22779.924,E2 -22779.924} C_VEL
LIN {X 0,Y 170.054,Z 535.195,A -85,B 0,C 180,E1 -22784.357,E2 -22784.357} C_VEL
LIN {X 0,Y 171.929,Z 530.639,A -85,B 0,C 180,E1 -22789.088,E2 -22789.088} C_VEL
LIN {X 0,Y 174.816,Z 524.63,A -85,B 0,C 180,E1 -22793.705,E2 -22793.705} C_VEL
LIN {X 0,Y 178.736,Z 517.014,A -85,B 0,C 180,E1 -22798.154,E2 -22798.154} C_VEL
LIN {X 0,Y 182.981,Z 508.81,A -85,B 0,C 180,E1 -22801.878,E2 -22801.878} C_VEL
LIN {X 0,Y 187.831,Z 498.905,A -85,B 0,C 180,E1 -22805.448,E2 -22805.448} C_VEL
LIN {X 0,Y 192.734,Z 488.72,A -85,B 0,C 180,E1 -22808.309,E2 -22808.309} C_VEL
LIN {X 0,Y 196.694,Z 479.771,A -85,B 0,C 180,E1 -22810.362,E2 -22810.362} C_VEL
LIN {X 0,Y 199.97,Z 471.863,A -85,B 0,C 180,E1 -22811.894,E2 -22811.894} C_VEL
LIN {X 0,Y 201.104,Z 460.125,A -85,B 0,C 180,E1 -22814.593,E2 -22814.593} C_VEL
LIN {X 0,Y 201.341,Z 448.295,A -85,B 0,C 180,E1 -22817.141,E2 -22817.141} C_VEL
LIN {X 0,Y 201.201,Z 445.503,A -85,B 0,C 180,E1 -22817.747,E2 -22817.747} C_VEL
LIN {X 0,Y 197.789,Z 434.376,A -85,B 0,C 180,E1 -22820.899,E2 -22820.899} C_VEL
LIN {X 0,Y 193.234,Z 423.224,A -85,B 0,C 180,E1 -22824.414,E2 -22824.414} C_VEL
LIN {X 0,Y 190.69,Z 418.211,A -85,B 0,C 180,E1 -22826.201,E2 -22826.201} C_VEL
LIN {X 0,Y 188.38,Z 413.663,A -85,B 0,C 180,E1 -22827.885,E2 -22827.885} C_VEL
LIN {X 0,Y 185.429,Z 408.526,A -85,B 0,C 180,E1 -22829.998,E2 -22829.998} C_VEL
LIN {X 0,Y 183,Z 404.524,A -85,B 0,C 180,E1 -22831.781,E2 -22831.781} C_VEL
LIN {X 0,Y 182.174,Z 403.035,A -85,B 0,C 180,E1 -22832.423,E2 -22832.423} C_VEL
LIN {X 0,Y 179.75,Z 399.869,A -85,B 0,C 180,E1 -22834.26,E2 -22834.26} C_VEL
LIN {X 0,Y 178.406,Z 397.157,A -85,B 0,C 180,E1 -22835.412,E2 -22835.412} C_VEL
LIN {X 0,Y 175.434,Z 394.134,A -85,B 0,C 180,E1 -22837.826,E2 -22837.826} C_VEL
LIN {X 0,Y 173.977,Z 391.185,A -85,B 0,C 180,E1 -22839.301,E2 -22839.301} C_VEL
LIN {X 0,Y 173.782,Z 390.554,A -85,B 0,C 180,E1 -22839.586,E2 -22839.586} C_VEL
LIN {X 0,Y 173.551,Z 389.026,A -85,B 0,C 180,E1 -22843.533,E2 -22843.533} C_VEL
LIN {X 0,Y 173.395,Z 387.521,A -85,B 0,C 180,E1 -22848.308,E2 -22848.308} C_VEL
LIN {X 0,Y 173.288,Z 386.418,A -85,B 0,C 180,E1 -22853.012,E2 -22853.012} C_VEL
LIN {X 0,Y 173.362,Z 385.632,A -85,B 0,C 180,E1 -22857.677,E2 -22857.677} C_VEL
LIN {X 0,Y 173.509,Z 385.341,A -85,B 0,C 180,E1 -22860,E2 -22860} C_VEL
LIN {X 0,Y 173.02,Z 385.231,A -85,B 0,C 180,E1 -22864.66,E2 -22864.66} C_VEL
LIN {X 0,Y 173.077,Z 385.353,A -85,B 0,C 180,E1 -22869.348,E2 -22869.348} C_VEL
LIN {X 0,Y 172.941,Z 385.902,A -85,B 0,C 180,E1 -22874.113,E2 -22874.113} C_VEL
LIN {X 0,Y 173.006,Z 386.768,A -85,B 0,C 180,E1 -22878.965,E2 -22878.965} C_VEL
LIN {X 0,Y 173.13,Z 387.809,A -85,B 0,C 180,E1 -22882.684,E2 -22882.684} C_VEL
LIN {X 0,Y 174.424,Z 390.471,A -85,B 0,C 180,E1 -22884.077,E2 -22884.077} C_VEL
LIN {X 0,Y 177.373,Z 393.365,A -85,B 0,C 180,E1 -22886.595,E2 -22886.595} C_VEL
LIN {X 0,Y 178.053,Z 394.23,A -85,B 0,C 180,E1 -22887.152,E2 -22887.152} C_VEL
LIN {X 0,Y 180.227,Z 397.798,A -85,B 0,C 180,E1 -22889.013,E2 -22889.013} C_VEL
LIN {X 0,Y 182.147,Z 399.963,A -85,B 0,C 180,E1 -22890.426,E2 -22890.426} C_VEL
LIN {X 0,Y 184.496,Z 403.744,A -85,B 0,C 180,E1 -22892.229,E2 -22892.229} C_VEL
LIN {X 0,Y 185.643,Z 405.361,A -85,B 0,C 180,E1 -22893.052,E2 -22893.052} C_VEL
LIN {X 0,Y 188.797,Z 410.877,A -85,B 0,C 180,E1 -22895.378,E2 -22895.378} C_VEL
LIN {X 0,Y 190.839,Z 414.484,A -85,B 0,C 180,E1 -22896.83,E2 -22896.83} C_VEL
LIN {X 0,Y 194.778,Z 422.867,A -85,B 0,C 180,E1 -22899.826,E2 -22899.826} C_VEL
LIN {X 0,Y 197.817,Z 431.134,A -85,B 0,C 180,E1 -22902.457,E2 -22902.457} C_VEL
LIN {X 0,Y 199.87,Z 440.543,A -85,B 0,C 180,E1 -22905.049,E2 -22905.049} C_VEL
LIN {X 0,Y 200.893,Z 450.379,A -85,B 0,C 180,E1 -22907.65,E2 -22907.65} C_VEL
LIN {X 0,Y 201.144,Z 460.005,A -85,B 0,C 180,E1 -22910.237,E2 -22910.237} C_VEL
LIN {X 0,Y 200.859,Z 462.801,A -85,B 0,C 180,E1 -22910.964,E2 -22910.964} C_VEL
LIN {X 0,Y 196.461,Z 473.29,A -85,B 0,C 180,E1 -22913.187,E2 -22913.187} C_VEL
LIN {X 0,Y 191.638,Z 483.766,A -85,B 0,C 180,E1 -22915.995,E2 -22915.995} C_VEL
LIN {X 0,Y 187.095,Z 492.479,A -85,B 0,C 180,E1 -22918.902,E2 -22918.902} C_VEL
LIN {X 0,Y 182.481,Z 500.879,A -85,B 0,C 180,E1 -22922.473,E2 -22922.473} C_VEL
LIN {X 0,Y 179.215,Z 506.813,A -85,B 0,C 180,E1 -22925.684,E2 -22925.684} C_VEL
LIN {X 0,Y 175.382,Z 513.191,A -85,B 0,C 180,E1 -22930.086,E2 -22930.086} C_VEL
LIN {X 0,Y 172.64,Z 518.007,A -85,B 0,C 180,E1 -22934.656,E2 -22934.656} C_VEL
LIN {X 0,Y 171.137,Z 520.728,A -85,B 0,C 180,E1 -22938.151,E2 -22938.151} C_VEL
LIN {X 0,Y 169.926,Z 523.172,A -85,B 0,C 180,E1 -22942.873,E2 -22942.873} C_VEL
LIN {X 0,Y 169.385,Z 524.386,A -85,B 0,C 180,E1 -22947.622,E2 -22947.622} C_VEL
LIN {X 0,Y 169.385,Z 524.404,A -85,B 0,C 180,E1 -22952.378,E2 -22952.378} C_VEL
LIN {X 0,Y 169.907,Z 523.229,A -85,B 0,C 180,E1 -22957.129,E2 -22957.129} C_VEL
LIN {X 0,Y 171.107,Z 520.825,A -85,B 0,C 180,E1 -22961.851,E2 -22961.851} C_VEL
LIN {X 0,Y 173.214,Z 517.111,A -85,B 0,C 180,E1 -22966.501,E2 -22966.501} C_VEL
LIN {X 0,Y 176.126,Z 511.985,A -85,B 0,C 180,E1 -22971.047,E2 -22971.047} C_VEL
LIN {X 0,Y 180.311,Z 505.221,A -85,B 0,C 180,E1 -22975.389,E2 -22975.389} C_VEL
LIN {X 0,Y 183.651,Z 498.981,A -85,B 0,C 180,E1 -22978.577,E2 -22978.577} C_VEL
LIN {X 0,Y 188.472,Z 490.154,A -85,B 0,C 180,E1 -22982.099,E2 -22982.099} C_VEL
LIN {X 0,Y 193.081,Z 480.969,A -85,B 0,C 180,E1 -22984.98,E2 -22984.98} C_VEL
LIN {X 0,Y 197.301,Z 471.847,A -85,B 0,C 180,E1 -22987.269,E2 -22987.269} C_VEL
LIN {X 0,Y 200.823,Z 463.394,A -85,B 0,C 180,E1 -22989.045,E2 -22989.045} C_VEL
LIN {X 0,Y 201.205,Z 460.467,A -85,B 0,C 180,E1 -22989.784,E2 -22989.784} C_VEL
LIN {X 0,Y 201.039,Z 450.81,A -85,B 0,C 180,E1 -22992.38,E2 -22992.38} C_VEL
LIN {X 0,Y 200.039,Z 441.155,A -85,B 0,C 180,E1 -22994.952,E2 -22994.952} C_VEL
LIN {X 0,Y 198.546,Z 433.542,A -85,B 0,C 180,E1 -22997.023,E2 -22997.023} C_VEL
LIN {X 0,Y 196.342,Z 426.694,A -85,B 0,C 180,E1 -22999.101,E2 -22999.101} C_VEL
LIN {X 0,Y 192.509,Z 417.78,A -85,B 0,C 180,E1 -23002.133,E2 -23002.133} C_VEL
LIN {X 0,Y 189.678,Z 412.499,A -85,B 0,C 180,E1 -23004.194,E2 -23004.194} C_VEL
LIN {X 0,Y 187.711,Z 408.785,A -85,B 0,C 180,E1 -23005.686,E2 -23005.686} C_VEL
LIN {X 0,Y 184.86,Z 404.168,A -85,B 0,C 180,E1 -23007.761,E2 -23007.761} C_VEL
LIN {X 0,Y 182.241,Z 400.181,A -85,B 0,C 180,E1 -23009.751,E2 -23009.751} C_VEL
LIN {X 0,Y 181.398,Z 398.966,A -85,B 0,C 180,E1 -23010.397,E2 -23010.397} C_VEL
LIN {X 0,Y 178.788,Z 395.723,A -85,B 0,C 180,E1 -23012.46,E2 -23012.46} C_VEL
LIN {X 0,Y 177.719,Z 393.602,A -85,B 0,C 180,E1 -23013.435,E2 -23013.435} C_VEL
LIN {X 0,Y 174.574,Z 390.682,A -85,B 0,C 180,E1 -23016.102,E2 -23016.102} C_VEL
LIN {X 0,Y 173.148,Z 387.943,A -85,B 0,C 180,E1 -23017.633,E2 -23017.633} C_VEL
LIN {X 0,Y 173.06,Z 387.581,A -85,B 0,C 180,E1 -23017.935,E2 -23017.935} C_VEL
LIN {X 0,Y 173.022,Z 386.871,A -85,B 0,C 180,E1 -23021.037,E2 -23021.037} C_VEL
LIN {X 0,Y 172.998,Z 385.822,A -85,B 0,C 180,E1 -23027.163,E2 -23027.163} C_VEL
LIN {X 0,Y 173.1,Z 385.456,A -85,B 0,C 180,E1 -23030.653,E2 -23030.653} C_VEL
LIN {X 0,Y 173.042,Z 385.338,A -85,B 0,C 180,E1 -23035.34,E2 -23035.34} C_VEL
LIN {X 0,Y 173.54,Z 385.419,A -85,B 0,C 180,E1 -23040,E2 -23040} C_VEL
LIN {X 0,Y 173.266,Z 386.088,A -85,B 0,C 180,E1 -23044.653,E2 -23044.653} C_VEL
LIN {X 0,Y 173.381,Z 387.003,A -85,B 0,C 180,E1 -23049.331,E2 -23049.331} C_VEL
LIN {X 0,Y 173.453,Z 388.311,A -85,B 0,C 180,E1 -23054.07,E2 -23054.07} C_VEL
LIN {X 0,Y 173.709,Z 390.017,A -85,B 0,C 180,E1 -23058.884,E2 -23058.884} C_VEL
LIN {X 0,Y 173.874,Z 390.753,A -85,B 0,C 180,E1 -23060.325,E2 -23060.325} C_VEL
LIN {X 0,Y 175.325,Z 393.928,A -85,B 0,C 180,E1 -23061.846,E2 -23061.846} C_VEL
LIN {X 0,Y 178.278,Z 397.052,A -85,B 0,C 180,E1 -23064.296,E2 -23064.296} C_VEL
LIN {X 0,Y 178.833,Z 397.947,A -85,B 0,C 180,E1 -23064.757,E2 -23064.757} C_VEL
LIN {X 0,Y 180.986,Z 401.755,A -85,B 0,C 180,E1 -23066.559,E2 -23066.559} C_VEL
LIN {X 0,Y 182.728,Z 403.761,A -85,B 0,C 180,E1 -23067.814,E2 -23067.814} C_VEL
LIN {X 0,Y 184.85,Z 407.743,A -85,B 0,C 180,E1 -23069.448,E2 -23069.448} C_VEL
LIN {X 0,Y 186.36,Z 409.991,A -85,B 0,C 180,E1 -23070.526,E2 -23070.526} C_VEL
LIN {X 0,Y 188.699,Z 414.093,A -85,B 0,C 180,E1 -23072.185,E2 -23072.185} C_VEL
LIN {X 0,Y 192.235,Z 421.189,A -85,B 0,C 180,E1 -23074.757,E2 -23074.757} C_VEL
LIN {X 0,Y 196.432,Z 430.787,A -85,B 0,C 180,E1 -23077.904,E2 -23077.904} C_VEL
LIN {X 0,Y 199.756,Z 440.347,A -85,B 0,C 180,E1 -23080.732,E2 -23080.732} C_VEL
LIN {X 0,Y 201.297,Z 445.773,A -85,B 0,C 180,E1 -23082.246,E2 -23082.246} C_VEL
LIN {X 0,Y 201.427,Z 455.094,A -85,B 0,C 180,E1 -23084.252,E2 -23084.252} C_VEL
LIN {X 0,Y 200.559,Z 468.018,A -85,B 0,C 180,E1 -23087.15,E2 -23087.15} C_VEL
LIN {X 0,Y 200.002,Z 472.131,A -85,B 0,C 180,E1 -23088.113,E2 -23088.113} C_VEL
LIN {X 0,Y 195.347,Z 483.141,A -85,B 0,C 180,E1 -23090.312,E2 -23090.312} C_VEL
LIN {X 0,Y 190.231,Z 494.219,A -85,B 0,C 180,E1 -23093.104,E2 -23093.104} C_VEL
LIN {X 0,Y 185.071,Z 504.766,A -85,B 0,C 180,E1 -23096.508,E2 -23096.508} C_VEL
LIN {X 0,Y 180.562,Z 513.812,A -85,B 0,C 180,E1 -23100.246,E2 -23100.246} C_VEL
LIN {X 0,Y 176.617,Z 521.143,A -85,B 0,C 180,E1 -23104.041,E2 -23104.041} C_VEL
LIN {X 0,Y 173.28,Z 527.906,A -85,B 0,C 180,E1 -23108.59,E2 -23108.59} C_VEL
LIN {X 0,Y 170.905,Z 533.151,A -85,B 0,C 180,E1 -23113.27,E2 -23113.27} C_VEL
LIN {X 0,Y 169.5,Z 537.011,A -85,B 0,C 180,E1 -23118.035,E2 -23118.035} C_VEL
LIN {X 0,Y 169.009,Z 539.568,A -85,B 0,C 180,E1 -23122.833,E2 -23122.833} C_VEL
LIN {X 0,Y 169.079,Z 540.858,A -85,B 0,C 180,E1 -23127.617,E2 -23127.617} C_VEL
LIN {X 0,Y 169.247,Z 541.027,A -85,B 0,C 180,E1 -23130,E2 -23130} C_VEL
LIN {X 0,Y 169.055,Z 540.357,A -85,B 0,C 180,E1 -23134.769,E2 -23134.769} C_VEL
LIN {X 0,Y 169.151,Z 538.412,A -85,B 0,C 180,E1 -23139.566,E2 -23139.566} C_VEL
LIN {X 0,Y 169.184,Z 538.197,A -85,B 0,C 180,E1 -23139.924,E2 -23139.924} C_VEL
LIN {X 0,Y 168.805,Z 537.031,A -85,B 0,C 180,E1 -23141.878,E2 -23141.878} C_VEL
LIN {X 0,Y 166.753,Z 534.687,A -85,B 0,C 180,E1 -23145.095,E2 -23145.095} C_VEL
LIN {X 0,Y 165.27,Z 532.48,A -85,B 0,C 180,E1 -23147.691,E2 -23147.691} C_VEL
LIN {X 0,Y 165.096,Z 530.561,A -85,B 0,C 180,E1 -23149.64,E2 -23149.64} C_VEL
LIN {X 0,Y 165.326,Z 529.872,A -85,B 0,C 180,E1 -23150.278,E2 -23150.278} C_VEL
LIN {X 0,Y 168.247,Z 524.273,A -85,B 0,C 180,E1 -23154.691,E2 -23154.691} C_VEL
LIN {X 0,Y 172.463,Z 516.654,A -85,B 0,C 180,E1 -23159.276,E2 -23159.276} C_VEL
LIN {X 0,Y 176.91,Z 508.44,A -85,B 0,C 180,E1 -23163.109,E2 -23163.109} C_VEL
LIN {X 0,Y 182.033,Z 498.525,A -85,B 0,C 180,E1 -23166.758,E2 -23166.758} C_VEL
LIN {X 0,Y 187.151,Z 488.323,A -85,B 0,C 180,E1 -23169.672,E2 -23169.672} C_VEL
LIN {X 0,Y 191.738,Z 478.275,A -85,B 0,C 180,E1 -23171.985,E2 -23171.985} C_VEL
LIN {X 0,Y 194.125,Z 472.519,A -85,B 0,C 180,E1 -23173.129,E2 -23173.129} C_VEL
LIN {X 0,Y 195.453,Z 460.65,A -85,B 0,C 180,E1 -23175.984,E2 -23175.984} C_VEL
LIN {X 0,Y 195.851,Z 450.008,A -85,B 0,C 180,E1 -23178.407,E2 -23178.407} C_VEL
LIN {X 0,Y 194.668,Z 444.518,A -85,B 0,C 180,E1 -23179.965,E2 -23179.965} C_VEL
LIN {X 0,Y 191.794,Z 435.461,A -85,B 0,C 180,E1 -23182.799,E2 -23182.799} C_VEL
LIN {X 0,Y 189.026,Z 428.219,A -85,B 0,C 180,E1 -23185.238,E2 -23185.238} C_VEL
LIN {X 0,Y 184.744,Z 419.214,A -85,B 0,C 180,E1 -23188.701,E2 -23188.701} C_VEL
LIN {X 0,Y 182.143,Z 414.245,A -85,B 0,C 180,E1 -23190.848,E2 -23190.848} C_VEL
LIN {X 0,Y 179.769,Z 409.902,A -85,B 0,C 180,E1 -23192.83,E2 -23192.83} C_VEL
LIN {X 0,Y 176.699,Z 405.144,A -85,B 0,C 180,E1 -23195.472,E2 -23195.472} C_VEL
LIN {X 0,Y 175.864,Z 403.398,A -85,B 0,C 180,E1 -23196.289,E2 -23196.289} C_VEL
LIN {X 0,Y 173.034,Z 400.021,A -85,B 0,C 180,E1 -23198.903,E2 -23198.903} C_VEL
LIN {X 0,Y 171.679,Z 397.041,A -85,B 0,C 180,E1 -23200.458,E2 -23200.458} C_VEL
LIN {X 0,Y 168.736,Z 394.234,A -85,B 0,C 180,E1 -23203.672,E2 -23203.672} C_VEL
LIN {X 0,Y 166.977,Z 391.118,A -85,B 0,C 180,E1 -23206.224,E2 -23206.224} C_VEL
LIN {X 0,Y 166.632,Z 389.962,A -85,B 0,C 180,E1 -23207.031,E2 -23207.031} C_VEL
LIN {X 0,Y 166.579,Z 389.121,A -85,B 0,C 180,E1 -23210.285,E2 -23210.285} C_VEL
LIN {X 0,Y 166.457,Z 388.189,A -85,B 0,C 180,E1 -23215.156,E2 -23215.156} C_VEL
LIN {X 0,Y 166.742,Z 387.475,A -85,B 0,C 180,E1 -23220,E2 -23220} C_VEL
LIN {X 0,Y 166.26,Z 387.356,A -85,B 0,C 180,E1 -23227.286,E2 -23227.286} C_VEL
LIN {X 0,Y 166.198,Z 387.726,A -85,B 0,C 180,E1 -23232.207,E2 -23232.207} C_VEL
LIN {X 0,Y 166.15,Z 388.259,A -85,B 0,C 180,E1 -23235.251,E2 -23235.251} C_VEL
LIN {X 0,Y 167.726,Z 391.35,A -85,B 0,C 180,E1 -23237.843,E2 -23237.843} C_VEL
LIN {X 0,Y 170.808,Z 394.086,A -85,B 0,C 180,E1 -23241.465,E2 -23241.465} C_VEL
LIN {X 0,Y 171.356,Z 394.76,A -85,B 0,C 180,E1 -23242.058,E2 -23242.058} C_VEL
LIN {X 0,Y 173.157,Z 397.941,A -85,B 0,C 180,E1 -23244.105,E2 -23244.105} C_VEL
LIN {X 0,Y 175.55,Z 400.378,A -85,B 0,C 180,E1 -23246.288,E2 -23246.288} C_VEL
LIN {X 0,Y 177.853,Z 404.263,A -85,B 0,C 180,E1 -23248.468,E2 -23248.468} C_VEL
LIN {X 0,Y 179.368,Z 406.227,A -85,B 0,C 180,E1 -23249.729,E2 -23249.729} C_VEL
LIN {X 0,Y 181.776,Z 410.151,A -85,B 0,C 180,E1 -23251.757,E2 -23251.757} C_VEL
LIN {X 0,Y 186.544,Z 419.046,A -85,B 0,C 180,E1 -23255.73,E2 -23255.73} C_VEL
LIN {X 0,Y 190.632,Z 428.394,A -85,B 0,C 180,E1 -23259.267,E2 -23259.267} C_VEL
LIN {X 0,Y 193.103,Z 436.116,A -85,B 0,C 180,E1 -23261.842,E2 -23261.842} C_VEL
LIN {X 0,Y 194.618,Z 444.869,A -85,B 0,C 180,E1 -23264.399,E2 -23264.399} C_VEL
LIN {X 0,Y 195.279,Z 454.978,A -85,B 0,C 180,E1 -23267.224,E2 -23267.224} C_VEL
LIN {X 0,Y 195.172,Z 463.25,A -85,B 0,C 180,E1 -23269.596,E2 -23269.596} C_VEL
LIN {X 0,Y 194.523,Z 465.546,A -85,B 0,C 180,E1 -23270.125,E2 -23270.125} C_VEL
LIN {X 0,Y 189.102,Z 477.406,A -85,B 0,C 180,E1 -23272.848,E2 -23272.848} C_VEL
LIN {X 0,Y 184.19,Z 487.224,A -85,B 0,C 180,E1 -23275.75,E2 -23275.75} C_VEL
LIN {X 0,Y 179.591,Z 495.442,A -85,B 0,C 180,E1 -23278.767,E2 -23278.767} C_VEL
LIN {X 0,Y 175.026,Z 503.343,A -85,B 0,C 180,E1 -23282.499,E2 -23282.499} C_VEL
LIN {X 0,Y 171.671,Z 508.94,A -85,B 0,C 180,E1 -23285.834,E2 -23285.834} C_VEL
LIN {X 0,Y 168.723,Z 513.541,A -85,B 0,C 180,E1 -23289.264,E2 -23289.264} C_VEL
LIN {X 0,Y 165.799,Z 518.354,A -85,B 0,C 180,E1 -23294.007,E2 -23294.007} C_VEL
LIN {X 0,Y 164.188,Z 521.074,A -85,B 0,C 180,E1 -23297.642,E2 -23297.642} C_VEL
LIN {X 0,Y 162.896,Z 523.517,A -85,B 0,C 180,E1 -23302.563,E2 -23302.563} C_VEL
LIN {X 0,Y 162.314,Z 524.731,A -85,B 0,C 180,E1 -23307.519,E2 -23307.519} C_VEL
LIN {X 0,Y 162.313,Z 524.748,A -85,B 0,C 180,E1 -23312.482,E2 -23312.482} C_VEL
LIN {X 0,Y 162.867,Z 523.574,A -85,B 0,C 180,E1 -23317.438,E2 -23317.438} C_VEL
LIN {X 0,Y 164.163,Z 521.17,A -85,B 0,C 180,E1 -23322.36,E2 -23322.36} C_VEL
LIN {X 0,Y 166.412,Z 517.456,A -85,B 0,C 180,E1 -23327.196,E2 -23327.196} C_VEL
LIN {X 0,Y 169.52,Z 512.333,A -85,B 0,C 180,E1 -23331.909,E2 -23331.909} C_VEL
LIN {X 0,Y 173.916,Z 505.576,A -85,B 0,C 180,E1 -23336.393,E2 -23336.393} C_VEL
LIN {X 0,Y 177.449,Z 499.335,A -85,B 0,C 180,E1 -23339.675,E2 -23339.675} C_VEL
LIN {X 0,Y 182.51,Z 490.52,A -85,B 0,C 180,E1 -23343.281,E2 -23343.281} C_VEL
LIN {X 0,Y 187.321,Z 481.346,A -85,B 0,C 180,E1 -23346.223,E2 -23346.223} C_VEL
LIN {X 0,Y 191.712,Z 472.244,A -85,B 0,C 180,E1 -23348.551,E2 -23348.551} C_VEL
LIN {X 0,Y 195.218,Z 463.828,A -85,B 0,C 180,E1 -23350.393,E2 -23350.393} C_VEL
